REGION Network 2: DESCRIPTION
   // The Energy Efficiency Monitor “EEM” integrated in SICAR is based on the application example in entry ID: 109753230 V1.0 dated 02/2018 of the Siemens Industry Online Support, see: 
   // 
   // https://support.industry.siemens.com/cs/document/109753230/-s7-energy-efficiency-monitor-for-machines?dti=0&lc=en-WW 
   // 
   // **License**  
   // The software package has to be licensed. The necessary license key has to be entered in the data block for energy data “EEmData”, in the array item “licenseKey”. 
   //  
   // {.pageWidth}
   // ![Image](EemEnPiCalc/en/image1.PNG)
   // 
   // The S7 Energy Efficiency-Monitor (or S7 EE-Monitor) allows you to record the energy consumption of your machine in a SIMATIC controller, and to analyze the results on the basis of the energy and media requirements.  
   // https://support.industry.siemens.com/cs/document/109753230/s7-energieeffizienz-monitor-für-maschinen?dti=0&lc=de-WW 
   // 
   // **PLC Data types**  
   //  LSicar_typeEeMenPiCalc 
   //  LSicar_typeEeMenPiEstate 
   //  LSicar_typeEeMenPiLimit 
   //  typeEnMeterOutputData 
   //  typeMeasDataProfileE3 
   //  
   // **WinCC Faceplates**  
   // 
   // ![Image](EemEnPiCalc/en/image3.PNG)
   // 
   // **WinCC Screen**  
   //  
   // ![Image](EemEnPiCalc/en/image4.PNG)
   //  
   // # Devices & networks 
   // 
   // An additional AI Energy Meter has been added and configured in the SICAR project. The user data has been  
   // configured as module version “EE@Industry measured data profile e3”.  
   // 
   // Select the module version according to your requirements. The data assignment in the FC blocks has to be adjusted according to the selected module version. 
   // 
   // ![Image](EemEnPiCalc/en/image5.PNG)
   //  
   //  
   // 
   //  #### PLC Programm blocks 
   // 
   // ##### CallEnSeem  
   // The block is called in OB “CYCLIC_INTERRUPT_100MS_OB” (100ms cycle). The block contains the following instructions which can be found in “Instructions > Optional packages > Energy Suite extensions”.
   // 
   // **EnS_EEm_Calc:**  
   // The instruction calculates operating state-related energy data of machines and plants for uniform efficiency evaluation, in accordance with the VDMA 34179 measuring directive. 
   // 
   // ---
   // Note
   // :     The instruction calculates the energy efficiency value of the respective state for up to 8 operating states, and the global energy efficiency value. 
   // :     The maximum number of configurable measuring points is 10. Refer to the documentation of the entry ID. 
   // 
   // ---
   // 
   // **EnS_EEm_Report:**  
   // The instruction writes the data for the efficiency report to the data log on the SIMATIC memory card, in accordance with the VDMA 34179 measuring directive. The data log is a CSV file. 
   // 
   // ##### CallEnEffMonitor
   // ---
   // Note
   // :     The assignment of the readings as well as the formation of additional signals can be represented only exemplarily here. It has to be adapted to the actual plant conditions! 
   // 
   // ---
   // 
   // * Networks 1 & 2: The readings of the two AI-Energy-Meters are entered in the DB “EeMonitor”, in an array [0..9] in accordance with the measurement data profile “typeMeasDataProfileE3”. 
   // * Network 3: According to the selection of a measuring point on the HMI, data of the respective measuring point is routed to the HMI data area. The selection is done with a Pull-Down menu and a symbolic I/O field. 
   // * Network 4: Several tags in the EnS…data types are not marked as accessible / visible. In order to display these tags on the HMI all the same, they are routed to DB “EeMonitor” in structure “typeEnMeterWorkHmi”. There the tags are marked as accessible / visible.  
   // * Network 5: A collective signal is generated, according to the exemplary calls for OP area 1. This is only an example! The collective signal shows that the plant is producing parts, by a disjunction (OR) of all outputs. If an output is controlled, the plant is moving and producing parts. This collective signal is used later on to generate the energetic states “eState”. A delay of 3 seconds has been configured so that a short break in controlling the outputs will not change the energetic state. *
   // * Network 6: The signals for the energetic states are generated here. 
   // * Network 7: Simulation On/Off: A part counter is simulated here. Note: the simulation can be switched on and off with a button in the screen. 
   // * Network 8: Simulation On/Off. Energy counters for both AI-Energy-Meters are simulated here. Note: the simulation can be switched on and off with a button in the screen. 
   // * Network 9: Call of blocks “EemDemoSimulation” and “EemDemoResetValEMeter”. 
   // * Network 10: Call of block “EemEnPiCalc” and data routing according to the selection of a measuring point on the HMI. 
   // * Network 11: Error evaluation of block “EemEnPiCalc” to generate ProDiag messages. 
   // * Network 12: Error evaluation of block “EnS_EEm_Report” to generate ProDiag messages.  
   // 
   // ##### EemDemoResetValEMeter  
   // 
   // The block resets certain measurement values by controlling the respective outputs in the I/O area of the AI-Energy-Meter. 
   // 
   // ##### EemDemoSimulation  
   // 
   // This block simulates higher or lower energy values, according to the energetic states “eState”. 
   // 
   // ##### EemEnPiCalc
   // This block calculates the ENPI (Energy value Pro Item). It substitutes the script “EEm_EnPI_Efficiency” of the entry ID. 
   // 
   // ---
   // Note
   // :     All block parameters are provided with “pre-defined actual parameters”.
   // 
   // ---
   // 
   // **Operation mode Automatic / Manual**  
   // 
   // The blocks are independent of operation modes. Therefor they are not assigned to any operation mode area. 
   // 
   // **PLC Alarm text list**  
   // 
   // The following PLC alarm text lists have been created: 
   // 
   // * **EEMonitor_Calc_Warn_PD** ProDiag alarm text list for alarms by instruction “EnS_EEm_Calc”.   
   // * **EEMonitor_Report_Warn_PD** ProDiag alarm text list for alarms by instruction “EnS_EEm_Report”.   
   // Both PLC alarm text lists have been entered in the PLC alarm text list “GLOBAL_GENERAL_AlarmTextList”. 
   // 
   // ---
   // Note
   // :     The alarm texts are provided in two languages (German, English). Please consider the multilingual nature of the entries. 
   // 
   // ---
   // 
   // #### PLC Data types 
   // 
   // PLC data types used for PLC program block or HMI faceplate:  
   // ![Image](_Icon/reference.PNG)  See ..\Library Types\LSicar_typeEeMenPiCalc.pdf  
   // 
   // #### WinCC Objects 
   // 
   // **WinCC HMI-tags**  
   // 
   // The HMI tags are stored in the tag table “AI_EnergyMeter_EEM” in the SICAR project.  
   // 
   // **WinCC Text and graphics lists**  
   // 
   // The text list “EE-MONITOR_MEASUREPOINT” contains the texts necessary for the pull-down menu / symbolic I/O field in the screen. Please take into account the multilingual nature of the entries.  
   // 
   // **WinCC Faceplates**  
   // 
   // The faceplates are stored in the project library, in folder “types”. They have been created using several WinCC objects; they are animated depending on the state. 
   // 
   // * EEM_EnPI_EnergyPerItem:	display of ENPI (ENergy Per Item) 
   // * EEM_ViewBar_Diff-AVG-REF:	bar display to compare reference value and average value 
   // * EEM_ViewBar_EState-Total:	bar display of energy status (not used at this time) 
   // * EEM_ViewBarCurve_EState:	Total: bar display and curve display of the energy values  
   // 
   // **WinCC-screen** 
   // 
   // 1. HMI Screens:	EE-MONITOR_ENERGY: display of the energy values 
   // 2. HMI Popup-screens 
   // 	* EEM_LEGEND_Popup: 		Legend 
   // 	* EEM_INFO-MACHINE_Popup: 	Machine information 
   // 	* EEM_STARTMEASURE_Popup: 	Popup to start the normal measurement or the reference measurement  
   // 	* EEM_UIPE_Popup: 		display of voltage, current, power, and energy 
   // 	* MORE_EEM_Popup: 		Popup with additional buttons 
   // 	* MORE_AddOn_Popup: 		supplemented  with button “EE-Monitor” 
   // 
   //  
   // 
   // {.pageWidth}
   // ![Image](EemEnPiCalc/en/image6.PNG)
   //  
   //  
   // 
   // #### Additional information
   // 
   // #### Update info
   // 
   // #### Further documentations
END_REGION

REGION Network 3: select measurement values
   // can be from EnergyMeter driver or directly from any hardware (in this example EnergyMeter module and PAC)
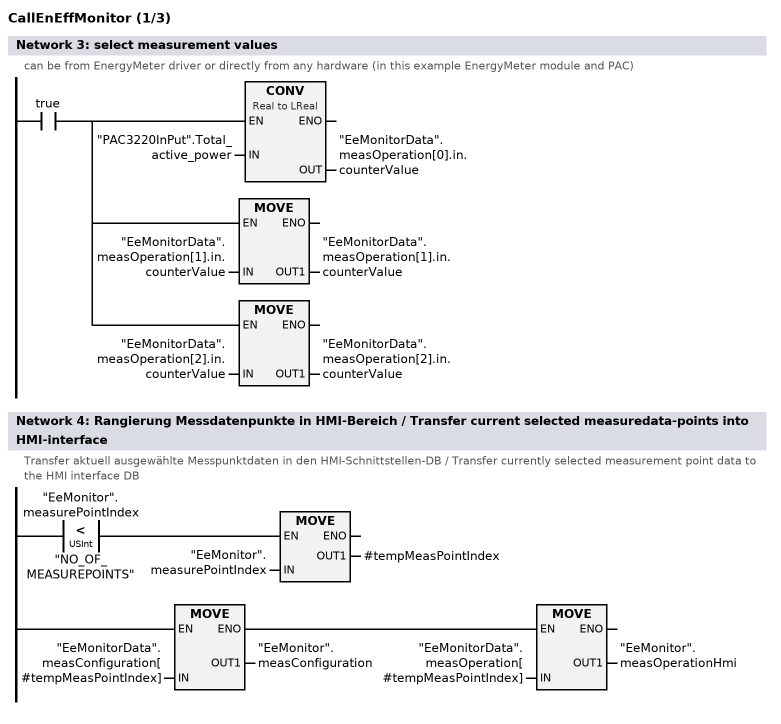
   RUNG wire#powerrail
      Contact( true )
      wire#w1
      { S7_Templates := "[SrcType := Real, DestType := LReal]" } Convert(in := "PAC3220InPut".Total_active_power, out => "EeMonitorData".measOperation[0].in.counterValue)
   END_RUNG
   RUNG wire#w1
      Move(in := "EeMonitorData".measOperation[1].in.counterValue, out1 => "EeMonitorData".measOperation[1].in.counterValue)
   END_RUNG
   RUNG wire#w1
      Move(in := "EeMonitorData".measOperation[2].in.counterValue, out1 => "EeMonitorData".measOperation[2].in.counterValue)
   END_RUNG
   // the same network as SCL:
   IF true THEN
       "EeMonitorData".measOperation[0].in.counterValue := REAL_TO_LREAL("PAC3220InPut".Total_active_power);
       "EeMonitorData".measOperation[1].in.counterValue := "EeMonitorData".measOperation[1].in.counterValue;
       "EeMonitorData".measOperation[2].in.counterValue := "EeMonitorData".measOperation[2].in.counterValue;
   END_IF;
END_REGION

REGION Network 4: Rangierung Messdatenpunkte in HMI-Bereich / Transfer current selected measuredata-points into HMI-interface
   // Transfer aktuell ausgewählte Messpunktdaten in den HMI-Schnittstellen-DB / Transfer currently selected measurement point data to the HMI interface DB
   RUNG wire#powerrail
      { S7_Templates := "SrcType := USInt" } LT_Contact(in1 := "EeMonitor".measurePointIndex, in2 := "NO_OF_MEASUREPOINTS")
      Move(in := "EeMonitor".measurePointIndex, out1 => #tempMeasPointIndex)
   END_RUNG
   RUNG wire#powerrail
      Move(in := "EeMonitorData".measConfiguration[#tempMeasPointIndex], out1 => "EeMonitor".measConfiguration)
      Move(in := "EeMonitorData".measOperation[#tempMeasPointIndex], out1 => "EeMonitor".measOperationHmi)
   END_RUNG
   // the same network as SCL:
   IF "EeMonitor".measurePointIndex < "NO_OF_MEASUREPOINTS" THEN
       #tempMeasPointIndex := "EeMonitor".measurePointIndex;
   END_IF;
   "EeMonitor".measConfiguration := "EeMonitorData".measConfiguration[#tempMeasPointIndex];
   "EeMonitor".measOperationHmi := "EeMonitorData".measOperation[#tempMeasPointIndex];
END_REGION

REGION Network 5: WORKaround: Rangierung / WORKaround: Transfer data from EeMonitroData to EeMonitor.work
   // Konvertierung Zeit in DTL und addieren Zeitzone mit Datum und Uhrzeit aus EnS_EEm_Calc zur Darstellung des tatsächlichen Datums und der tatsächlichen Uhrzeit im aktuellen Land.
   // Convertion of Time to DTL and adding time zone with date and time taken from EnS_EEm_Calc for representing the actual date and time in the current country.
   // Data is copied from EeMonitorData to EeMonitor.work
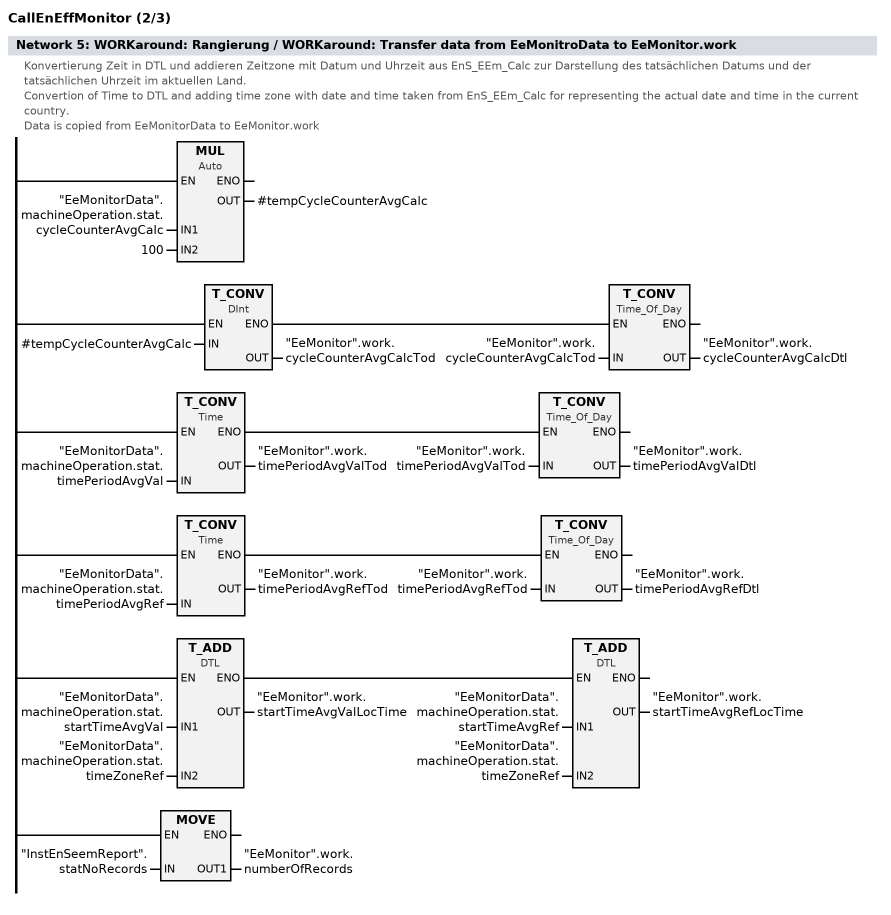
   RUNG wire#powerrail
      Mul(in1 := "EeMonitorData".machineOperation.stat.cycleCounterAvgCalc, in2 := 100, out => #tempCycleCounterAvgCalc)
   END_RUNG
   RUNG wire#powerrail
      { S7_Templates := "[src_type := DInt, dest_type := Time_Of_Day]" } T_CONV(IN := #tempCycleCounterAvgCalc, OUT => "EeMonitor".work.cycleCounterAvgCalcTod)
      { S7_Templates := "[src_type := Time_Of_Day, dest_type := DTL]" } T_CONV(IN := "EeMonitor".work.cycleCounterAvgCalcTod, OUT => "EeMonitor".work.cycleCounterAvgCalcDtl)
   END_RUNG
   RUNG wire#powerrail
      { S7_Templates := "[src_type := Time, dest_type := Time_Of_Day]" } T_CONV(IN := "EeMonitorData".machineOperation.stat.timePeriodAvgVal, OUT => "EeMonitor".work.timePeriodAvgValTod)
      { S7_Templates := "[src_type := Time_Of_Day, dest_type := DTL]" } T_CONV(IN := "EeMonitor".work.timePeriodAvgValTod, OUT => "EeMonitor".work.timePeriodAvgValDtl)
   END_RUNG
   RUNG wire#powerrail
      { S7_Templates := "[src_type := Time, dest_type := Time_Of_Day]" } T_CONV(IN := "EeMonitorData".machineOperation.stat.timePeriodAvgRef, OUT => "EeMonitor".work.timePeriodAvgRefTod)
      { S7_Templates := "[src_type := Time_Of_Day, dest_type := DTL]" } T_CONV(IN := "EeMonitor".work.timePeriodAvgRefTod, OUT => "EeMonitor".work.timePeriodAvgRefDtl)
   END_RUNG
   RUNG wire#powerrail
      { S7_Templates := "[date_type := DTL, time_type := Time]" } T_ADD(IN1 := "EeMonitorData".machineOperation.stat.startTimeAvgVal, IN2 := "EeMonitorData".machineOperation.stat.timeZoneRef, OUT => "EeMonitor".work.startTimeAvgValLocTime)
      { S7_Templates := "[date_type := DTL, time_type := Time]" } T_ADD(IN1 := "EeMonitorData".machineOperation.stat.startTimeAvgRef, IN2 := "EeMonitorData".machineOperation.stat.timeZoneRef, OUT => "EeMonitor".work.startTimeAvgRefLocTime)
   END_RUNG
   RUNG wire#powerrail
      Move(in := "InstEnSeemReport".statNoRecords, out1 => "EeMonitor".work.numberOfRecords)
   END_RUNG
   // the same network as SCL:
   #tempCycleCounterAvgCalc := "EeMonitorData".machineOperation.stat.cycleCounterAvgCalc * 100;
   T_CONV(IN := #tempCycleCounterAvgCalc, OUT => "EeMonitor".work.cycleCounterAvgCalcTod, ENO => #_w1);
   IF #_w1 THEN
       T_CONV(IN := "EeMonitor".work.cycleCounterAvgCalcTod, OUT => "EeMonitor".work.cycleCounterAvgCalcDtl);
   END_IF;
   T_CONV(IN := "EeMonitorData".machineOperation.stat.timePeriodAvgVal,
          OUT => "EeMonitor".work.timePeriodAvgValTod,
          ENO => #_w2);
   IF #_w2 THEN
       T_CONV(IN := "EeMonitor".work.timePeriodAvgValTod, OUT => "EeMonitor".work.timePeriodAvgValDtl);
   END_IF;
   T_CONV(IN := "EeMonitorData".machineOperation.stat.timePeriodAvgRef,
          OUT => "EeMonitor".work.timePeriodAvgRefTod,
          ENO => #_w3);
   IF #_w3 THEN
       T_CONV(IN := "EeMonitor".work.timePeriodAvgRefTod, OUT => "EeMonitor".work.timePeriodAvgRefDtl);
   END_IF;
   T_ADD(IN1 := "EeMonitorData".machineOperation.stat.startTimeAvgVal,
         IN2 := "EeMonitorData".machineOperation.stat.timeZoneRef,
         OUT => "EeMonitor".work.startTimeAvgValLocTime,
         ENO => #_w4);
   IF #_w4 THEN
       T_ADD(IN1 := "EeMonitorData".machineOperation.stat.startTimeAvgRef,
             IN2 := "EeMonitorData".machineOperation.stat.timeZoneRef,
             OUT => "EeMonitor".work.startTimeAvgRefLocTime);
   END_IF;
   "EeMonitor".work.numberOfRecords := "InstEnSeemReport".statNoRecords;
END_REGION

REGION Network 6: Betriebsarten für BA-Bereich1 auf "eState" in "EEm_Data_DB" / Operation modes to "eState"
   // Setzt Estate Nummer abhängig vom ausgewählten OpMode1-Modus / Sets Estate number accoriding to the selected state
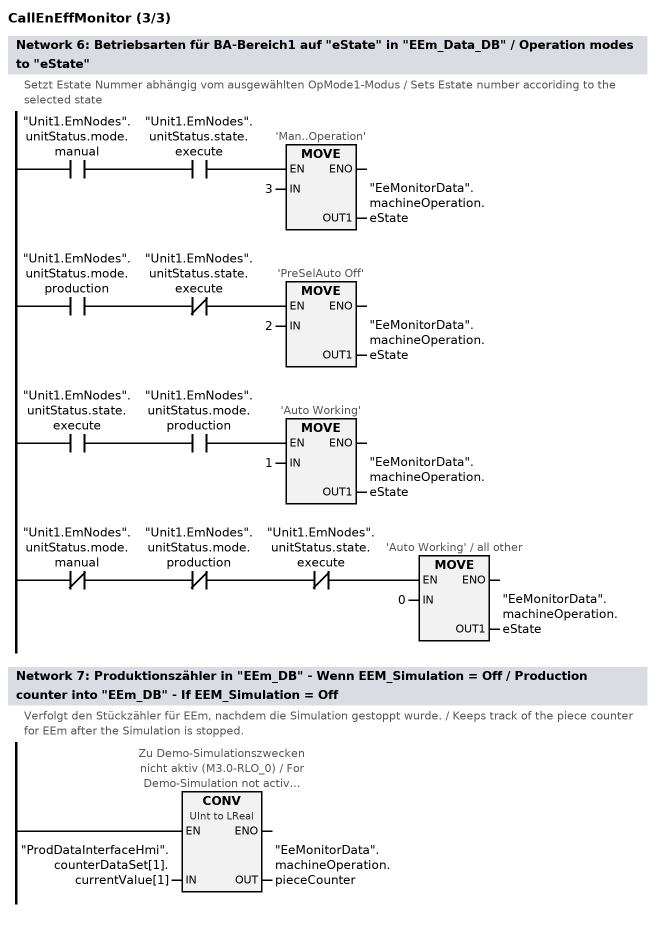
   RUNG wire#powerrail
      Contact( "Unit1.EmNodes".unitStatus.mode.manual )
      Contact( "Unit1.EmNodes".unitStatus.state.execute )
      Move(in := 3, out1 => "EeMonitorData".machineOperation.eState)   // 'Man..Operation'
   END_RUNG
   RUNG wire#powerrail
      Contact( "Unit1.EmNodes".unitStatus.mode.production )
      I_Contact( "Unit1.EmNodes".unitStatus.state.execute )
      Move(in := 2, out1 => "EeMonitorData".machineOperation.eState)   // 'PreSelAuto Off'
   END_RUNG
   RUNG wire#powerrail
      Contact( "Unit1.EmNodes".unitStatus.state.execute )
      Contact( "Unit1.EmNodes".unitStatus.mode.production )
      Move(in := 1, out1 => "EeMonitorData".machineOperation.eState)   // 'Auto Working'
   END_RUNG
   RUNG wire#powerrail
      I_Contact( "Unit1.EmNodes".unitStatus.mode.manual )
      I_Contact( "Unit1.EmNodes".unitStatus.mode.production )
      I_Contact( "Unit1.EmNodes".unitStatus.state.execute )
      Move(in := 0, out1 => "EeMonitorData".machineOperation.eState)   // 'Auto Working' / all other
   END_RUNG
   // the same network as SCL:
   IF "Unit1.EmNodes".unitStatus.mode.manual AND "Unit1.EmNodes".unitStatus.state.execute THEN
       "EeMonitorData".machineOperation.eState := 3;   // 'Man..Operation'
   END_IF;
   IF "Unit1.EmNodes".unitStatus.mode.production AND NOT "Unit1.EmNodes".unitStatus.state.execute THEN
       "EeMonitorData".machineOperation.eState := 2;   // 'PreSelAuto Off'
   END_IF;
   IF "Unit1.EmNodes".unitStatus.state.execute AND "Unit1.EmNodes".unitStatus.mode.production THEN
       "EeMonitorData".machineOperation.eState := 1;   // 'Auto Working'
   END_IF;
   IF NOT "Unit1.EmNodes".unitStatus.mode.manual AND NOT "Unit1.EmNodes".unitStatus.mode.production AND NOT "Unit1.EmNodes".unitStatus.state.execute THEN
       "EeMonitorData".machineOperation.eState := 0;   // 'Auto Working' / all other
   END_IF;
END_REGION

REGION Network 7: Produktionszähler in "EEm_DB" - Wenn EEM_Simulation = Off / Production counter into "EEm_DB" - If EEM_Simulation = Off
   // Verfolgt den Stückzähler für EEm, nachdem die Simulation gestoppt wurde. / Keeps track of the piece counter for EEm after the Simulation is stopped.
   RUNG wire#powerrail
      { S7_Templates := "[SrcType := UInt, DestType := LReal]" } Convert(in := "ProdDataInterfaceHmi".counterDataSet[1].currentValue[1], out => "EeMonitorData".machineOperation.pieceCounter)   // Zu Demo-Simulationszwecken nicht aktiv (M3.0-RLO_0) / For Demo-Simulation not active (M3.0-RLO_0)
   END_RUNG
   // the same network as SCL:
   "EeMonitorData".machineOperation.pieceCounter := UINT_TO_LREAL("ProdDataInterfaceHmi".counterDataSet[1].currentValue[1]);   // Zu Demo-Simulationszwecken nicht aktiv (M3.0-RLO_0) / For Demo-Simulation not active (M3.0-RLO_0)
END_REGION

REGION Network 8 (SCL): Temporary value for storing the EnPi reset time / Reset EnPI values
   // Liest die aktuelle Uhrzeit und speichert sie, um dem Benutzer Informationen über den letzten EnPi-Reset bereitzustellen / Reads the current time and store it to provide the user the information about the last EnPi reset
   // Check for the trigger to reset/recalculate the EnPI values
   IF ("EeMonitorData".internalData.enpiResetTrigger = TRUE) THEN

       // Read the current time and store it to provide the user the information
       // about the last reset
       #tempReturnValue := RD_LOC_T("EeMonitorData".internalData.enpiResetTime);

       // Reset the trigger
       "EeMonitorData".internalData.enpiResetTrigger := FALSE;
   ELSE
       ; // No trigger
   END_IF;
END_REGION
END_FUNCTION

FUNCTION "CallSettings" : Void   // FC8, LAD
// Call of settings blocks
// stored: IsIECCheckEnabled true, SetENOAutomatically false
BEGIN

REGION Network 1: Beschreibung / BLOCK INFO HEADER
   // **Betriebsart Automatik / Hand**  
   // Der Baustein ist keiner Betriebsart / Betriebsartenbereich zugeordnet.  
   // 
   // **Alarme**  
   // Der Baustein generiert keine Alarme.  
   // 
   // #### PLC-Datentypen  
   // Verwendete PLC-Datentypen für den SPS-Programmbaustein und das zugehörige WinCC-Bild.  
   // 
   // {.pageWidth}
   // ![Image](CallInterfaceSignals/de/image1.PNG)
   //  
   //  
   // #### Bausteinaufrufe 
   // Der Baustein “LSicar_InterfaceSignalsBool“ wird in diesem FB als Multi-Instanz aufgerufen, entspr. nebenstehender beispielhafter Darstellung.  
   // 
   // {.pageWidth}
   // ![Image](CallInterfaceSignals/de/image2.PNG)
   //  
   // Um einen neuen FB aufzurufen, ziehen Sie den FB in ein neues Netzwerk, wählen Sie „Multiinstanz“ aus, vergeben Sie einen Namen und parametrieren Sie den FB-Aufruf.  
   // 
   // {.pageWidth}
   // ![Image](CallInterfaceSignals/de/image3.PNG)
   //  
   //  
   // #### Weitere Hinweise 
   // 
   // #### Updateinfo 
   // 
   // #### Weitere Dokumente 
   // 
   // ![Icon](_Icon/reference.PNG)
   // 
   // ..\Library Types\LSicar_InterfaceSignalsBool.pdf
   // SIEMENS AG / (c)Copyright 2023
   // ------------------------------------------------------------------------------
   // Title:            CallSettings
   // Comment/Function: Call of SICAR Settings blocks
   // Library/Family:   -
   // Author:           -
   // Tested with:      ---
   // Engineering:      TIA Portal V19
   // Restrictions:     -
   // Requirements:     ---
   // ------------------------------------------------------------------------------
   // Change log table:
   // Version | Date | Expert in charge | Changes applied
   // -------|---------|-------------|--------------------------------------------
   // 01.00.00 | 01.01.1999 | Person x | First released version
   // 01.00.01 | 02.01.1999 | Person y | Block was Updated
END_REGION

REGION Network 2: Set set PLC date and time
   // Change local date and time of the PLC
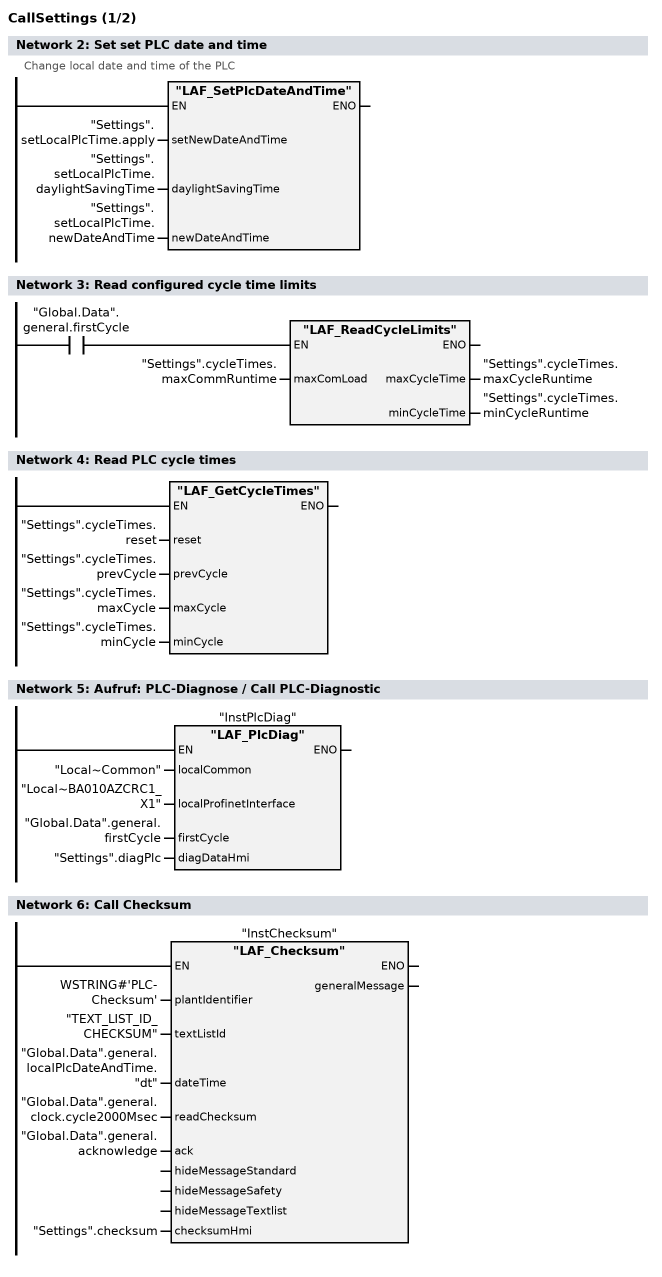
   RUNG wire#powerrail
      "LAF_SetPlcDateAndTime"(setNewDateAndTime := "Settings".setLocalPlcTime.apply, daylightSavingTime := "Settings".setLocalPlcTime.daylightSavingTime, newDateAndTime := "Settings".setLocalPlcTime.newDateAndTime)
   END_RUNG
   // the same network as SCL:
   "LAF_SetPlcDateAndTime"(setNewDateAndTime := "Settings".setLocalPlcTime.apply,
                           daylightSavingTime := "Settings".setLocalPlcTime.daylightSavingTime,
                           newDateAndTime := "Settings".setLocalPlcTime.newDateAndTime);
END_REGION

REGION Network 3: Read configured cycle time limits
   RUNG wire#powerrail
      Contact( "Global.Data".general.firstCycle )
      "LAF_ReadCycleLimits"(maxComLoad := "Settings".cycleTimes.maxCommRuntime, maxCycleTime => "Settings".cycleTimes.maxCycleRuntime, minCycleTime => "Settings".cycleTimes.minCycleRuntime)
   END_RUNG
   // the same network as SCL:
   IF "Global.Data".general.firstCycle THEN
       "LAF_ReadCycleLimits"(maxComLoad := "Settings".cycleTimes.maxCommRuntime,
                             maxCycleTime => "Settings".cycleTimes.maxCycleRuntime,
                             minCycleTime => "Settings".cycleTimes.minCycleRuntime);
   END_IF;
END_REGION

REGION Network 4: Read PLC cycle times
   RUNG wire#powerrail
      "LAF_GetCycleTimes"(reset := "Settings".cycleTimes.reset, prevCycle := "Settings".cycleTimes.prevCycle, maxCycle := "Settings".cycleTimes.maxCycle, minCycle := "Settings".cycleTimes.minCycle)
   END_RUNG
   // the same network as SCL:
   "LAF_GetCycleTimes"(reset := "Settings".cycleTimes.reset,
                       prevCycle := "Settings".cycleTimes.prevCycle,
                       maxCycle := "Settings".cycleTimes.maxCycle,
                       minCycle := "Settings".cycleTimes.minCycle);
END_REGION

REGION Network 5: Aufruf: PLC-Diagnose / Call PLC-Diagnostic
   RUNG wire#powerrail
      "InstPlcDiag"(localCommon := "Local~Common", localProfinetInterface := "Local~BA010AZCRC1_X1", firstCycle := "Global.Data".general.firstCycle, diagDataHmi := "Settings".diagPlc)
   END_RUNG
   // the same network as SCL:
   "InstPlcDiag"(localCommon := "Local~Common",   // "LAF_PlcDiag"
                 localProfinetInterface := "Local~BA010AZCRC1_X1",
                 firstCycle := "Global.Data".general.firstCycle,
                 diagDataHmi := "Settings".diagPlc);
END_REGION

REGION Network 6: Call Checksum
   RUNG wire#powerrail
      "InstChecksum"(plantIdentifier := WSTRING#'PLC-Checksum', textListId := "TEXT_LIST_ID_CHECKSUM", dateTime := "Global.Data".general.localPlcDateAndTime."dt", readChecksum := "Global.Data".general.clock.cycle2000Msec, ack := "Global.Data".general.acknowledge, hideMessageStandard :=, hideMessageSafety :=, hideMessageTextlist :=, checksumHmi := "Settings".checksum, generalMessage =>)
   END_RUNG
   // the same network as SCL:
   "InstChecksum"(plantIdentifier := WSTRING#'PLC-Checksum',   // "LAF_Checksum"
                  textListId := "TEXT_LIST_ID_CHECKSUM",
                  dateTime := "Global.Data".general.localPlcDateAndTime."dt",
                  readChecksum := "Global.Data".general.clock.cycle2000Msec,
                  ack := "Global.Data".general.acknowledge,
                  checksumHmi := "Settings".checksum);
END_REGION

REGION Network 7: Aufruf: SMC-Diagnose (SIMATIC Memory Card - Diagnose) / Call SMC-Diagnostic (SIMATIC Memory Card - Diagnostic)
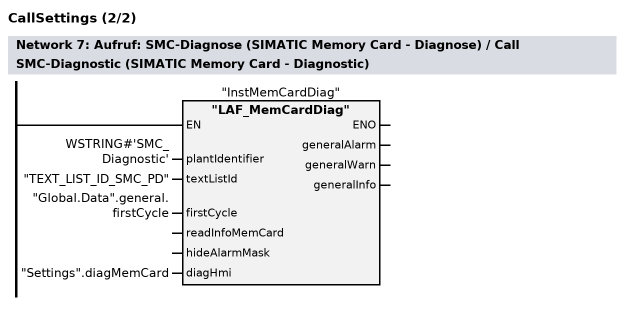
   RUNG wire#powerrail
      "InstMemCardDiag"(plantIdentifier := WSTRING#'SMC_Diagnostic', textListId := "TEXT_LIST_ID_SMC_PD", firstCycle := "Global.Data".general.firstCycle, readInfoMemCard :=, hideAlarmMask :=, diagHmi := "Settings".diagMemCard, generalAlarm =>, generalWarn =>, generalInfo =>)
   END_RUNG
   // the same network as SCL:
   "InstMemCardDiag"(plantIdentifier := WSTRING#'SMC_Diagnostic',   // "LAF_MemCardDiag"
                     textListId := "TEXT_LIST_ID_SMC_PD",
                     firstCycle := "Global.Data".general.firstCycle,
                     diagHmi := "Settings".diagMemCard);
END_REGION
END_FUNCTION

ORGANIZATION_BLOCK "Interrupt1s"   // OB31, LAD, CyclicInterrupt
TITLE = Zyklischer Interrupt 100ms / Cyclic interrupt 100ms
AUTHOR : SICAR
FAMILY : OB
VERSION : 1.0
// organisation block
// stored: IsIECCheckEnabled true, SetENOAutomatically true
   VAR_INPUT
      Initial_Call : Bool;   // Initial call of this OB
      Event_Count : Int;   // Events discarded
   END_VAR
BEGIN

REGION Network 1: Änderungshistorie / ChangeLog
   // Die Änderungshistorie wird nur in englischer Editiersprache geführt.
   // Change log table:
   // Version | Date | Expert in charge | Changes applied
   // -------|---------|-------------|--------------------------------------------
   // 01.00.00 | 01.01.1999 | Person x | First released version
   // 01.00.01 | 02.01.1999 | Person y | Block was Updated
END_REGION

REGION Network 2: EE-MONITOR: Aufruf & Mess-Daten in "EEmData_DB" / Call & measure-data into "EEmData_DB"
   // Aufruf der Energieeffizienz Überwachungs Functionen / Call the energy efficiency monitor functions
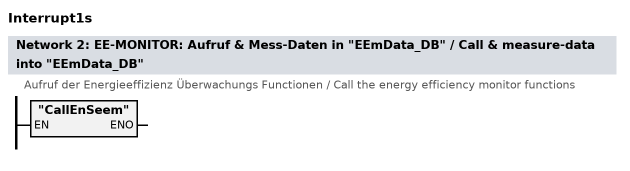
   RUNG wire#powerrail
      "CallEnSeem"()
   END_RUNG
   // the same network as SCL:
   "CallEnSeem"();
END_REGION
END_ORGANIZATION_BLOCK

FUNCTION "CallEnSeem" : Void   // FC34, LAD
TITLE = CallEnSeem
AUTHOR : SICAR
FAMILY : Energy_EEM
VERSION : 1.0
// Der in SICAR eingebaute Energie Effizienz Monitor „EEM“ basiert auf der Beitrags-ID: 109753230, V1.0 von 02/2018 des Siemens Industry Online Support, siehe:  
// https://support.industry.siemens.com/cs/document/109753230/s7-energieeffizienz-monitor-f%C3%BCr-maschinen?dti=0&lc=de-WW  
// 
// **Lizenz**  
// Das Softwarepaket ist Lizenzpflichtig. Die notwendige Lizenz muss im Datenbaustein der Energiedaten „EeMonitorData“ im Datum „licencsKey“ eingetragen werden.  
// 
// 
// Mit dem S7 Energieeffizienz-Monitor können Sie Energieverbräuche Ihrer Maschine in einer SIMATIC Steuerung erfassen und anhand des Energie- und Medienbedarfs statusbezogen anhand der energetischen Zustände analy-sieren. 
//  
//  
// **SPS-Programmbausteine**  
//  
// **PLC-Datentypen**  
//   LSicar_typeEeMenPiCalc  
//   LSicar_typeEeMenPiEstate  
//   LSicar_typeEeMenPiLimit  
//   typeEnMeterOutputData  
//   typeMeasDataProfileE3  
// 
// **WinCC-Bildbaustein**  
//  
// **WinCC-Bild**  
//  
//  
// #### Geräte & Netze
// Im SICAR-Projekt ist ein weiteres AI Energy Meter eingefügt und konfiguriert. Dies ist unter „Nutzdaten“ mit der Modulversion „EE@Industry Messdatenprofil e3“ parametriert.  
// Wählen Sie entsprechend Ihren Anforderungen die Modulversion aus. Je nach gewählter Modulversion, muss die Datenrangierung in den FC-Bausteinen angepasst werden.  
//  
// 
// #### SPS-Programmbausteine
// **CallEnSeem**  
// Der Baustein wird im OB „CYCLIC_INTERRUPT_100MS_OB“ (100ms Takt) aufgerufen. Darin sind nachfolgende Baustein-Anweisungen. Sie sind enthalten unter „Optionspakete > Energy Suite Erweiterungen“.  
// 
// **EnS_EEm_Calc:**  
// Der Baustein berechnet betriebszustandsbezogene Energiedaten von Maschinen und Anlagen zur einheitlichen Effizienzbewertung gemäß Messvorschrift VDMA 34179.  
// 
// NOTE
//  
// :     Der Baustein berechnet für bis zu acht Betriebszustände den Energieeffizienzwert des jeweiligen Zustands sowie den Gesamt-Energieeffizienzwert. 
// :     Die maximale Anzahl der konfigurierbaren Messstellen ist 10. Beachten Sie hierzu die Dokumentation der Beitrags-ID.
// 
// ---
// 
// **EnS_EEm_Report:**  
// Der Baustein erstellt ein Effizienzprotokoll im CSV-Format auf der SIMATIC Memory Card der CPU gemäß Messvorschrift VDMA 34179.  
// 
// **CallEnEffMonitor**  
// 
// NOTE
// :     Die Rangierung der Messdaten, sowie die Bildung von zusätzlichen Signalen kann hier nur beispiel-haft dargestellt werden. Sie muss auf die tatsächlichen Anlagengegebenheiten angepasst werden!
// 
// ---
// 
// * **Netzwerk 1 & 2:** In den beiden Netzwerken werden die Messdaten der beiden AI-Energy-Meter in den DB „EeMonitor“ einge-tragen, in ein Arrayfeld [0..9] gemäß dem Messdatenprofil " typeMeasDataProfileE3".
// * **Netzwerk 3:** Entsprechend des auf dem HMI angewählten Messpunktes (Pull-Down-Menü / Symbolisches E/A-Feld) wer-den hier die Daten des jeweiligen Messpunktes in dem HMI-Datenbereich rangiert.
// * **Netzwerk 4:** Einige Daten in den EnS…-Datentypen (im DB „EeMonitorData“) sind nicht mit Erreichbar/Sichtbar gekenn-zeichnet. Um diese Daten dennoch auf dem HMI darzustellen, werden sie in dem DB „EeMonitor“ rangiert in die Struktur „typeEnMeterWorkHmi“; dort sind die Daten mit Erreichbar/Sichtbar gekennzeichnet. 
// * **Netzwerk 5:** Hier wird ein Summensignal gebildet, entsprechend den Beispiel-Aufrufen für Betriebsartenbereich 1. Es han-delt sich hierbei lediglich um eine Beispiel-Anwendung! Das Summensignal gibt an, das die Anlage Teile pro-duziert. Hierzu werden alle Ausgänge verodert: Werden die Ausgänge angesteuert, so bewegt sich die Anla-ge, die Anlage produziert. Dieses Summensignal wird später benötigt, um damit die energetischen Zustände „eState“ zu bilden. Damit eine kurze Pause bzgl. der Ansteuerung der Ausgänge nicht zu einem Wechsel des energetischen Zustands führt ist hier eine Zeitverzögerung von 3 Sekunden eingebaut.
// * **Netzwerk 6:** In diesem Netzwerk werden die Signale für die energetischen Zustände gebildet.
// * **Netzwerk 7:** Simulation Ein/Aus Betrifft die Simulation von einem Stückzähler. Es wird hier ein simulierter Zähler als Stückzähler verwendet. Hinweis: Die Simulation kann im Bild mittels eines Buttons ein- und ausgeschaltet werden.
// * **Netzwerk 8:** Simulation Ein/Aus Betrifft die Simulation von Energiezähler für beide AI-Energy-Meter. Hinweis: Die Simulation kann im Bild mittels eines Button Ein- und Ausgeschaltet werden.
// * **Netzwerk 9:** Aufruf der Bausteine „EemDemoSimulation“ und „“EemDemoResetValEmeter“.
// * **Netzwerk 10:** Aufruf des Bausteins „EemEnPiCalc“ und Rangierung der daten entspr. dem auf dem HMI ausgewählten Messpunktes.
// * **Netzwerk 11:** Fehlerauswertung des Bausteins “ EemEnPiCalc“ zur Generierung von ProDiag-Meldungen.
// * **Netzwerk 12:** Fehlerauswertung des Bausteins “EnS_EEm_Report“ zur Generierung von ProDiag-Meldungen.
// 
// **EemDemoResetValEmeter** Der Baustein führt ein Reset auf gewisse Messwerte aus, durch Zuweisen der entspr. Ausgänge im E/A-Bereich der AI-Energy-Meter.
// **EemDemoSimulation** Baustein zur Simulation von höheren oder niedrigeren Energiewerten entsprechend der energetischen Zustände „eState“.
// **EemEnPiCalc** Der Baustein berechnet den ENPI (Energiewert Pro Item). Er ersetzt das Skript „EEm_EnPI_Efficiency“ der Bei-trags-ID.
// 
// **Parameter**  
// 
// NOTE
// :     Alle Bausteinparameter sind mit "Vordefinierten Aktualparametern" versehen.
// 
// ---
// 
// **Betriebsart Automatik / Hand** 
// Die Bausteine sind keinem Betriebsartenbereich zugeordnet.  
// 
// **PLC-Meldetextliste**  
// Folgende PLC-Meldetextlisten wurden hierzu angelegt:  
// * EEMonitor_Calc_Warn_PD Beinhaltet die ProDiag-Meldetext für den Bausteinaufruf „EnS_EEm_Calc“.  
// * EEMonitor_Report_Warn_PD Beinhaltet die ProDiag-Meldetexte für den Bausteinaufruf „EnS_EEm_Report“  
// 
// Beide Meldetextlisten sind in der PLC-Meldetextliste „GLOBAL_GENERAL_AlarmTextList“ eingetragen.  
// 
// NOTE
// :    Die Textlisten sind in Deutsch und Englisch ausgeführt. Bitte beachten Sie die Mehrsprachigkeit der PLC-Meldetextlisten.
// 
// ---
// 
// #### PLC-Datentypen
// Verwendete PLC-Datentypen für den SPS-Programmbaustein / WinCC-Bildbaustein:  
// Siehe ..\Library Types\LSicar_typeEeMenPiCalc.pdf  
//  
// #### WinCC-Objekte
// **WinCC HMI-Variablen**  
// Die HMI-Variablen sind im SICAR-Projekt angelegt in der Variablentabelle „AI_EnergyMeter_EEM“  
// 
// **WinCC Text- und Grafiklisten**  
// Die für das im Bild befindliche Pull-Down-Menü / Symbolisches E/A-Feld notwendigen Texte sind in der Text- und Grafikliste „EE-MONITOR_MEASUREPOINT“ hinterlegt. Bitte beachten Sie auch hier die Mehrsprachigkeit.  
// 
// **WinCC-Bildbaustein**  
// Die Bildbausteine befinden sich in der Projekt-Bibliothek unter „Typen“. Sie sind erstellt aus mehreren einzelnen WinCC-Objekten und animiert, je nach Zustand.  
// * EEM_EnPI_EnergyPerItem: Darstellung ENPI (Energy Per Item)
// * EEM_ViewBar_Diff-AVG-REF: Balkendarstellung zum Vergleich zwischen Referenz- / Durchschnittswert
// * EEM_ViewBar_EState-Total: Balkendarstellung Energie Status (z.Zt. nicht verwendet)
// * EEM_ViewBarCurve_EState-Total: Balken- und Kurvendarstellung der Energiewerte
// 
// **WinCC-Bild**  
// * HMI Bilder	
// 	- EE-MONITOR_ENERGY: Darstellung der Energiewerte
// * HMI Popup-Bilder	
// 	- EEM_LEGEND_Popup: Legende
// 	- EEM_INFO-MACHINE_Popup: Maschineninformationen
// 	- EEM_STARTMEASURE_Popup: Popup zum Starten der Normal- oder Referenzmessung
// 	- EEM_UIPE_Popup: Darstellung von Spannung, Strom, Leistung und Energie
// 	- MORE_EEM_Popup: Popup mit zusätzlichen Schaltflächen / Buttons
// 	- MORE_AddOn_Popup: Ergänzt um Button „EE-Monitor“
//  
// #### Weitere Hinweise
// 
// #### Updateinfo
// 
// #### Weitere Dokumente
// The S7 Energy Efficiency-Monitor (or S7 EE-Monitor) allows you to record the energy consumption of your machine in a SIMATIC controller, and to analyze the results on the basis of the energy and media requirements.
// stored: IsIECCheckEnabled true, SetENOAutomatically true
   // Ret_Val : Ret_Val
BEGIN

REGION Network 1: Änderungshistorie / BLOCK INFO HEADER
   // Die Änderungshistorie wird nur in englischer Editiersprache geführt.
   // SIEMENS AG / (c)Copyright 2023
   // ------------------------------------------------------------------------------
   // Title:            CallEnSeem (FC34)
   // Comment/Function: The S7 Energy Efficiency-Monitor (or S7 EE-Monitor) allows you to record the energy consumption of your machine in a SIMATIC controller, and to analyze the results on the basis of the energy and media requirements.
   // Library/Family:   Energy_EEM
   // Author:           SICAR
   // Tested with:      ---
   // Engineering:      TIA Portal V19
   // Restrictions:     -
   // Requirements:     ---
   // ------------------------------------------------------------------------------
   // Change log table:
   // Version | Date | Expert in charge | Changes applied
   // -------|---------|-------------|--------------------------------------------
   // 01.00.00 | 01.01.1999 | Person x | First released version
   // 01.00.01 | 02.01.1999 | Person y | Block was Updated
END_REGION

REGION Network 2: DESCRIPTION
   // The Energy Efficiency Monitor “EEM” integrated in SICAR is based on the application example in entry ID: 109753230 V1.0 dated 02/2018 of the Siemens Industry Online Support, see: 
   // 
   // https://support.industry.siemens.com/cs/document/109753230/-s7-energy-efficiency-monitor-for-machines?dti=0&lc=en-WW 
   // 
   // **License**  
   // The software package has to be licensed. The necessary license key has to be entered in the data block for energy data “EEmData”, in the array item “licenseKey”. 
   //  
   // {.pageWidth}
   // ![Image](EemEnPiCalc/en/image1.PNG)
   // 
   // The S7 Energy Efficiency-Monitor (or S7 EE-Monitor) allows you to record the energy consumption of your machine in a SIMATIC controller, and to analyze the results on the basis of the energy and media requirements.  
   // https://support.industry.siemens.com/cs/document/109753230/s7-energieeffizienz-monitor-für-maschinen?dti=0&lc=de-WW 
   // 
   // **PLC Data types**  
   //  LSicar_typeEeMenPiCalc 
   //  LSicar_typeEeMenPiEstate 
   //  LSicar_typeEeMenPiLimit 
   //  typeEnMeterOutputData 
   //  typeMeasDataProfileE3 
   //  
   // **WinCC Faceplates**  
   // 
   // ![Image](EemEnPiCalc/en/image3.PNG)
   // 
   // **WinCC Screen**  
   //  
   // ![Image](EemEnPiCalc/en/image4.PNG)
   //  
   // # Devices & networks 
   // 
   // An additional AI Energy Meter has been added and configured in the SICAR project. The user data has been  
   // configured as module version “EE@Industry measured data profile e3”.  
   // 
   // Select the module version according to your requirements. The data assignment in the FC blocks has to be adjusted according to the selected module version. 
   // 
   // ![Image](EemEnPiCalc/en/image5.PNG)
   //  
   //  
   // 
   // #### PLC Programm blocks 
   // 
   // ##### CallEnSeem  
   // The block is called in OB “CYCLIC_INTERRUPT_100MS_OB” (100ms cycle). The block contains the following instructions which can be found in “Instructions > Optional packages > Energy Suite extensions”.
   // 
   // **EnS_EEm_Calc:**  
   // The instruction calculates operating state-related energy data of machines and plants for uniform efficiency evaluation, in accordance with the VDMA 34179 measuring directive. 
   // 
   // ---
   // Note
   // :     The instruction calculates the energy efficiency value of the respective state for up to 8 operating states, and the global energy efficiency value. 
   // :     The maximum number of configurable measuring points is 10. Refer to the documentation of the entry ID. 
   // 
   // ---
   // 
   // **EnS_EEm_Report:**  
   // The instruction writes the data for the efficiency report to the data log on the SIMATIC memory card, in accordance with the VDMA 34179 measuring directive. The data log is a CSV file. 
   // 
   // #### CallEnEffMonitor
   // ---
   // Note
   // :     The assignment of the readings as well as the formation of additional signals can be represented only exemplarily here. It has to be adapted to the actual plant conditions! 
   // 
   // ---
   // 
   // * Networks 1 & 2: The readings of the two AI-Energy-Meters are entered in the DB “EeMonitor”, in an array [0..9] in accordance with the measurement data profile “typeMeasDataProfileE3”. 
   // * Network 3: According to the selection of a measuring point on the HMI, data of the respective measuring point is routed to the HMI data area. The selection is done with a Pull-Down menu and a symbolic I/O field. 
   // * Network 4: Several tags in the EnS…data types are not marked as accessible / visible. In order to display these tags on the HMI all the same, they are routed to DB “EeMonitor” in structure “typeEnMeterWorkHmi”. There the tags are marked as accessible / visible.  
   // * Network 5: A collective signal is generated, according to the exemplary calls for OP area 1. This is only an example! The collective signal shows that the plant is producing parts, by a disjunction (OR) of all outputs. If an output is controlled, the plant is moving and producing parts. This collective signal is used later on to generate the energetic states “eState”. A delay of 3 seconds has been configured so that a short break in controlling the outputs will not change the energetic state. *
   // * Network 6: The signals for the energetic states are generated here. 
   // * Network 7: Simulation On/Off: A part counter is simulated here. Note: the simulation can be switched on and off with a button in the screen. 
   // * Network 8: Simulation On/Off. Energy counters for both AI-Energy-Meters are simulated here. Note: the simulation can be switched on and off with a button in the screen. 
   // * Network 9: Call of blocks “EemDemoSimulation” and “EemDemoResetValEMeter”. 
   // * Network 10: Call of block “EemEnPiCalc” and data routing according to the selection of a measuring point on the HMI. 
   // * Network 11: Error evaluation of block “EemEnPiCalc” to generate ProDiag messages. 
   // * Network 12: Error evaluation of block “EnS_EEm_Report” to generate ProDiag messages.  
   // 
   // #### EemDemoResetValEMeter  
   // 
   // The block resets certain measurement values by controlling the respective outputs in the I/O area of the AI-Energy-Meter. 
   // 
   // #### EemDemoSimulation  
   // 
   // This block simulates higher or lower energy values, according to the energetic states “eState”. 
   // 
   // #### EemEnPiCalc
   // This block calculates the ENPI (Energy value Pro Item). It substitutes the script “EEm_EnPI_Efficiency” of the entry ID. 
   // 
   // ---
   // Note
   // :     All block parameters are provided with “pre-defined actual parameters”.
   // 
   // ---
   // 
   // **Operation mode Automatic / Manual**  
   // 
   // The blocks are independent of operation modes. Therefor they are not assigned to any operation mode area. 
   // 
   // **PLC Alarm text list**  
   // 
   // The following PLC alarm text lists have been created: 
   // 
   // * **EEMonitor_Calc_Warn_PD** ProDiag alarm text list for alarms by instruction “EnS_EEm_Calc”.   
   // * **EEMonitor_Report_Warn_PD** ProDiag alarm text list for alarms by instruction “EnS_EEm_Report”.   
   // Both PLC alarm text lists have been entered in the PLC alarm text list “GLOBAL_GENERAL_AlarmTextList”. 
   // 
   // ---
   // Note
   // :     The alarm texts are provided in two languages (German, English). Please consider the multilingual nature of the entries. 
   // 
   // ---
   // 
   // #### PLC Data types 
   // 
   // PLC data types used for PLC program block or HMI faceplate:  
   // ![Image](_Icon/reference.PNG)  See ..\Library Types\LSicar_typeEeMenPiCalc.pdf  
   // 
   // #### WinCC Objects 
   // 
   // **WinCC HMI-tags**  
   // 
   // The HMI tags are stored in the tag table “AI_EnergyMeter_EEM” in the SICAR project.  
   // 
   // **WinCC Text and graphics lists**  
   // 
   // The text list “EE-MONITOR_MEASUREPOINT” contains the texts necessary for the pull-down menu / symbolic I/O field in the screen. Please take into account the multilingual nature of the entries.  
   // 
   // **WinCC Faceplates**  
   // 
   // The faceplates are stored in the project library, in folder “types”. They have been created using several WinCC objects; they are animated depending on the state. 
   // 
   // * EEM_EnPI_EnergyPerItem:	display of ENPI (ENergy Per Item) 
   // * EEM_ViewBar_Diff-AVG-REF:	bar display to compare reference value and average value 
   // * EEM_ViewBar_EState-Total:	bar display of energy status (not used at this time) 
   // * EEM_ViewBarCurve_EState:	Total: bar display and curve display of the energy values  
   // 
   // **WinCC-screen** 
   // 
   // 1. HMI Screens:	EE-MONITOR_ENERGY: display of the energy values 
   // 2. HMI Popup-screens 
   // 	* EEM_LEGEND_Popup: 		Legend 
   // 	* EEM_INFO-MACHINE_Popup: 	Machine information 
   // 	* EEM_STARTMEASURE_Popup: 	Popup to start the normal measurement or the reference measurement  
   // 	* EEM_UIPE_Popup: 		display of voltage, current, power, and energy 
   // 	* MORE_EEM_Popup: 		Popup with additional buttons 
   // 	* MORE_AddOn_Popup: 		supplemented  with button “EE-Monitor” 
   // 
   //  
   // 
   // {.pageWidth}
   // ![Image](EemEnPiCalc/en/image6.PNG)
   //  
   //  
   // 
   // #### Additional information
   // 
   // #### Update info
   // 
   // #### Further documentations
END_REGION

REGION Network 3: EE-Monitor: "Recalc"
   // Toggeln für autom. Aktualisierung der Werte im Bild jeden zweiten Zyklus (alle 200ms) / Toggle for autom. updating the values in the screen every 2nd cycle (every 200ms)
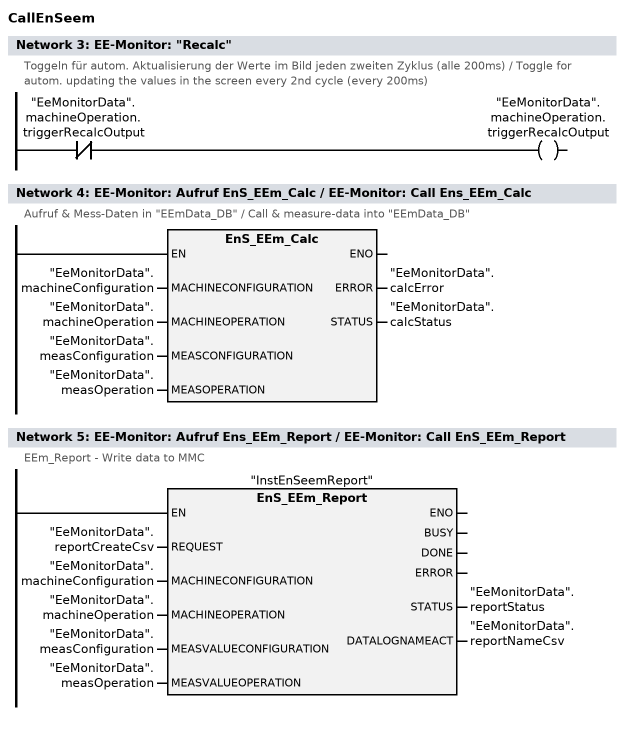
   RUNG wire#powerrail
      I_Contact( "EeMonitorData".machineOperation.triggerRecalcOutput )
      Coil( "EeMonitorData".machineOperation.triggerRecalcOutput )
   END_RUNG
   // the same network as SCL:
   "EeMonitorData".machineOperation.triggerRecalcOutput := NOT "EeMonitorData".machineOperation.triggerRecalcOutput;
END_REGION

REGION Network 4: EE-Monitor: Aufruf EnS_EEm_Calc / EE-Monitor: Call Ens_EEm_Calc
   // Aufruf & Mess-Daten in "EEmData_DB" / Call & measure-data into "EEmData_DB"
   RUNG wire#powerrail
      EnS_EEm_Calc(machineConfiguration := "EeMonitorData".machineConfiguration, machineOperation := "EeMonitorData".machineOperation, measConfiguration := "EeMonitorData".measConfiguration, measOperation := "EeMonitorData".measOperation, error => "EeMonitorData".calcError, status => "EeMonitorData".calcStatus)
   END_RUNG
   // the same network as SCL:
   EnS_EEm_Calc(machineConfiguration := "EeMonitorData".machineConfiguration,
                machineOperation := "EeMonitorData".machineOperation,
                measConfiguration := "EeMonitorData".measConfiguration,
                measOperation := "EeMonitorData".measOperation,
                error => "EeMonitorData".calcError,
                status => "EeMonitorData".calcStatus);
END_REGION

REGION Network 5: EE-Monitor: Aufruf Ens_EEm_Report / EE-Monitor: Call EnS_EEm_Report
   // EEm_Report - Write data to MMC
   RUNG wire#powerrail
      "InstEnSeemReport".EnS_EEm_Report(request := "EeMonitorData".reportCreateCsv, machineConfiguration := "EeMonitorData".machineConfiguration, machineOperation := "EeMonitorData".machineOperation, measValueConfiguration := "EeMonitorData".measConfiguration, measValueOperation := "EeMonitorData".measOperation, busy =>, done =>, error =>, status => "EeMonitorData".reportStatus, dataLogNameAct => "EeMonitorData".reportNameCsv)
   END_RUNG
   // the same network as SCL:
   "InstEnSeemReport"(request := "EeMonitorData".reportCreateCsv,   // EnS_EEm_Report
                      machineConfiguration := "EeMonitorData".machineConfiguration,
                      machineOperation := "EeMonitorData".machineOperation,
                      measValueConfiguration := "EeMonitorData".measConfiguration,
                      measValueOperation := "EeMonitorData".measOperation,
                      status => "EeMonitorData".reportStatus,
                      dataLogNameAct => "EeMonitorData".reportNameCsv);
END_REGION
END_FUNCTION

ORGANIZATION_BLOCK "ProgrammingError"   // OB121, LAD, ProgrammingError
// stored: SetENOAutomatically false
   VAR_INPUT
      BlockNr : UInt;   // Number of causing block
      Reaction : USInt;   // 0:ignore, 1:substitute, 2:skip
      Fault_ID : Byte;   // Fault identifier
      BlockType : USInt;   // 16#01:OB, 16#02:FC, 16#03:FB, 16#04:SFC, 16#05:SFB, 16#06:DB: Type of block causing the error
      Area : USInt;   // Area where the error occured
      DBNr : DB_ANY;   // DB number if Area = DB or DI
      Csg_OBNr : OB_ANY;   // Number of OB causing the error
      Csg_Prio : USInt;   // Priority of OB causing the error
      Width : USInt;   // 0:bit, 1:byte, 2:word, 3:dword, 4:lword
   END_VAR
BEGIN
END_ORGANIZATION_BLOCK

ORGANIZATION_BLOCK "Startup"   // OB100, LAD, Startup
TITLE = "Complete Restart"
// stored: AutoNumber false, IsIECCheckEnabled true, SetENOAutomatically true
   VAR_INPUT
      LostRetentive : Bool;   // True if retentive data are lost
      LostRTC : Bool;   // True if date and time are lost
   END_VAR
   VAR_TEMP
      tempError : Bool;
      tempStatus : Word;
      tempDiagnostics : "LAF_typeDiagnosticsSimple";
   END_VAR
BEGIN

REGION Network 1: Erster Zyklus bit setzen / Set first cycle bit
   // Setze das "erster Zyklus" Signal und die Signale immer EIN sowie immer AUS / Set the first cycle signal
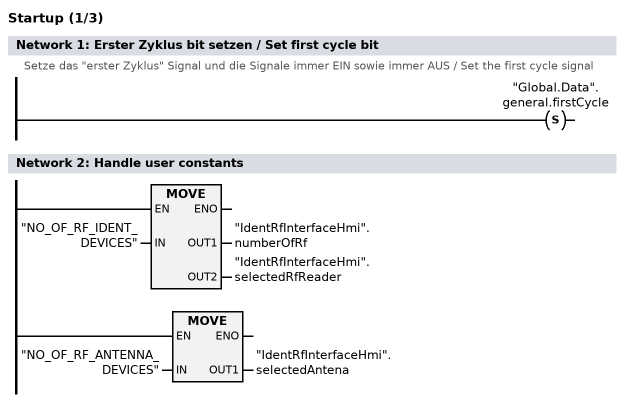
   RUNG wire#powerrail
      S_Coil( "Global.Data".general.firstCycle )
   END_RUNG
   // the same network as SCL:
   "Global.Data".general.firstCycle := TRUE;
END_REGION

REGION Network 2: Handle user constants
   RUNG wire#powerrail
      Move(in := "NO_OF_RF_IDENT_DEVICES", out1 => "IdentRfInterfaceHmi".numberOfRf, out2 => "IdentRfInterfaceHmi".selectedRfReader)
   END_RUNG
   RUNG wire#powerrail
      Move(in := "NO_OF_RF_ANTENNA_DEVICES", out1 => "IdentRfInterfaceHmi".selectedAntena)
   END_RUNG
   // the same network as SCL:
   "IdentRfInterfaceHmi".numberOfRf := "NO_OF_RF_IDENT_DEVICES";
   "IdentRfInterfaceHmi".selectedRfReader := "NO_OF_RF_IDENT_DEVICES";
   "IdentRfInterfaceHmi".selectedAntena := "NO_OF_RF_ANTENNA_DEVICES";
END_REGION

REGION Network 3: Set drive objects for drive diagnostic
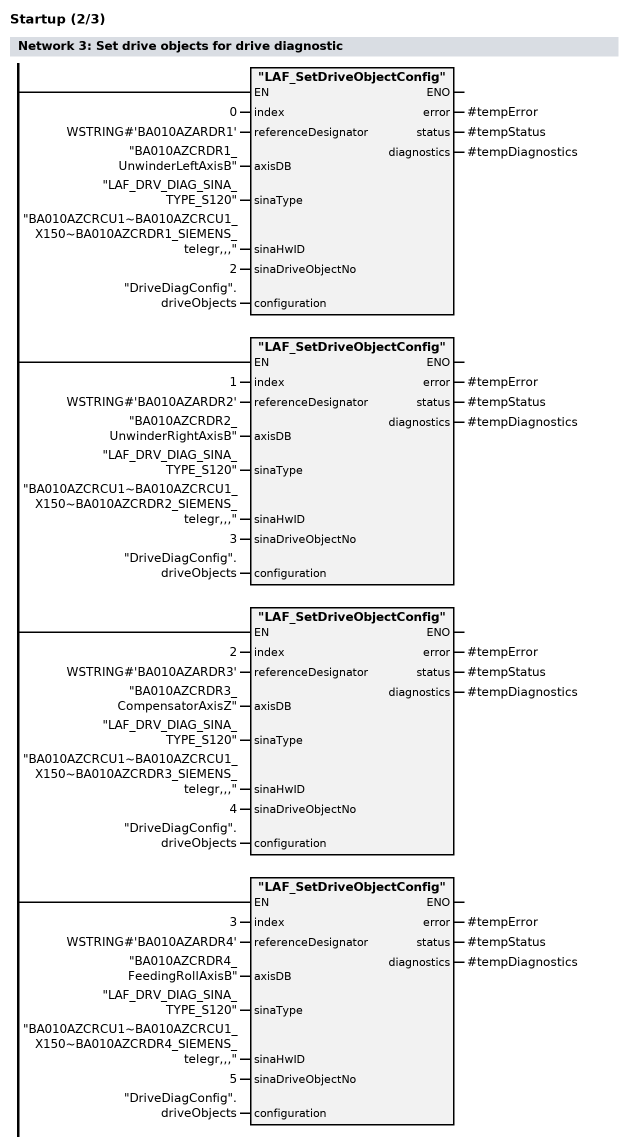
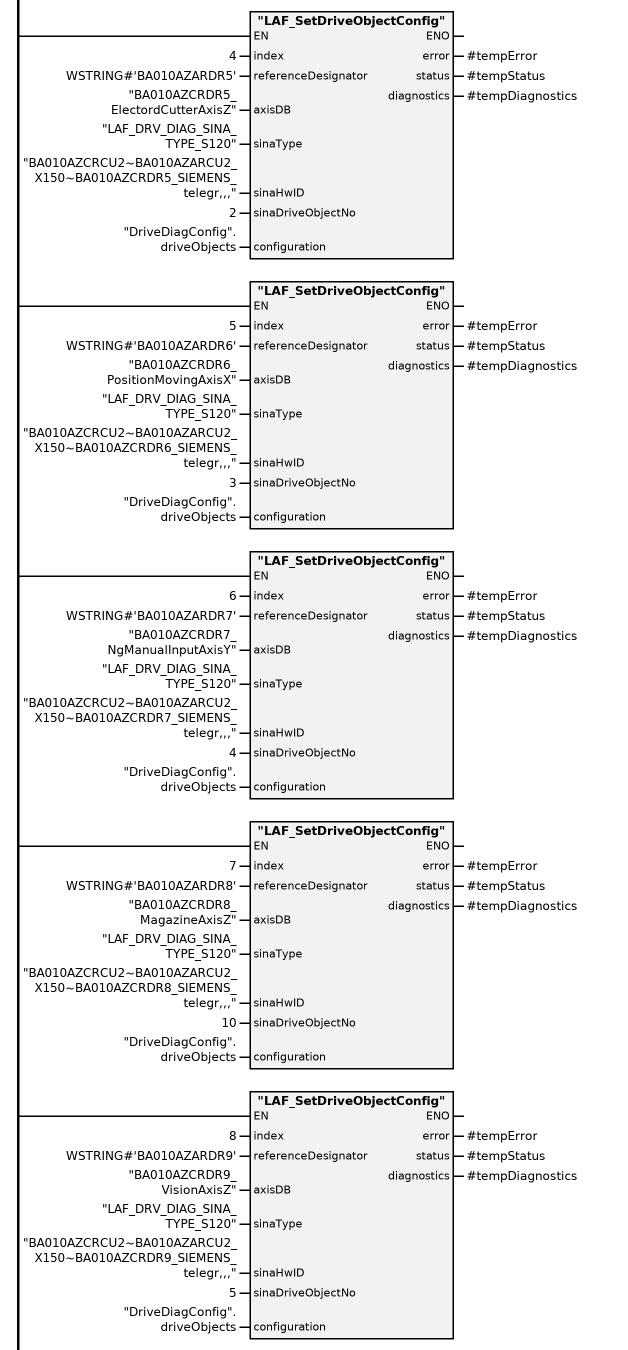
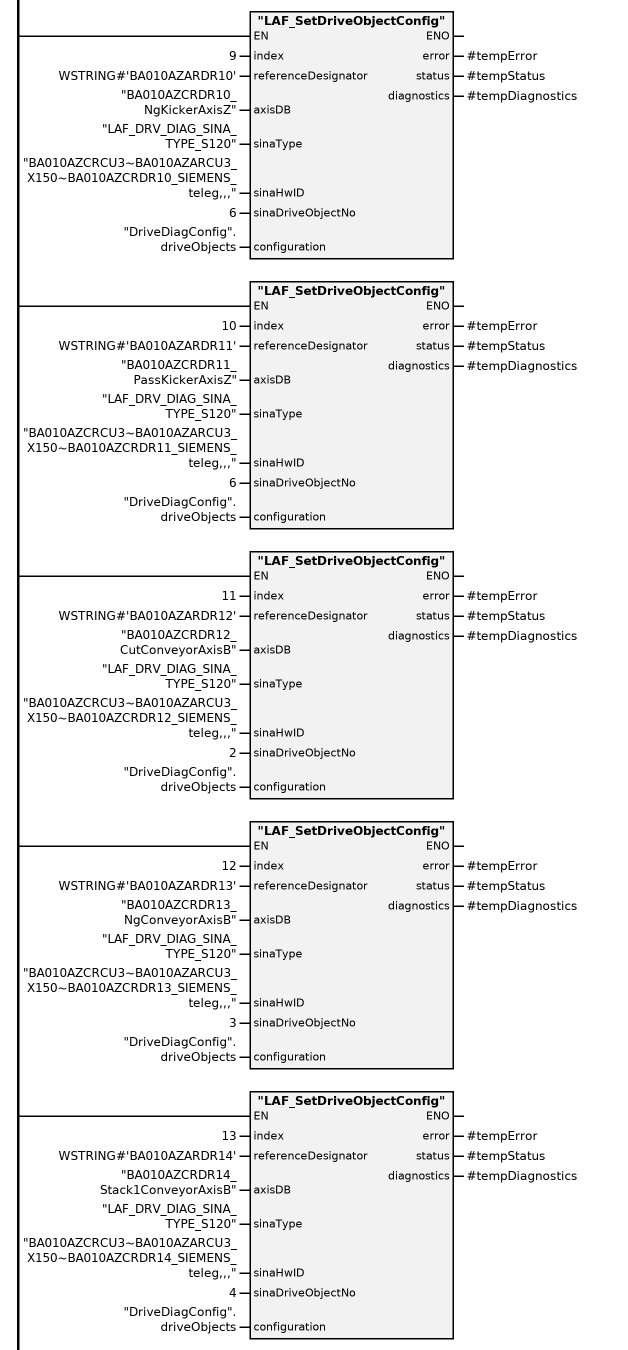
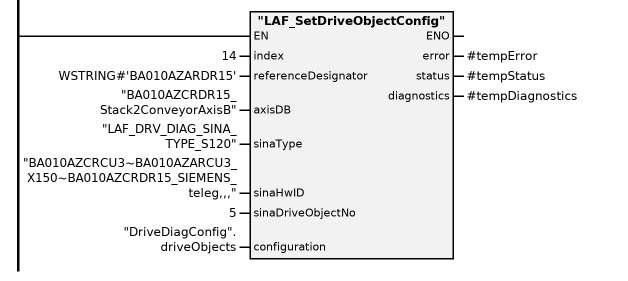
   RUNG wire#powerrail
      "LAF_SetDriveObjectConfig"(index := 0, referenceDesignator := WSTRING#'BA010AZARDR1', axisDB := "BA010AZCRDR1_UnwinderLeftAxisB", sinaType := "LAF_DRV_DIAG_SINA_TYPE_S120", sinaHwID := "BA010AZCRCU1~BA010AZCRCU1_X150~BA010AZCRDR1_SIEMENS_telegr,,,", sinaDriveObjectNo := 2, configuration := "DriveDiagConfig".driveObjects, error => #tempError, status => #tempStatus, diagnostics => #tempDiagnostics)
   END_RUNG
   RUNG wire#powerrail
      "LAF_SetDriveObjectConfig"(index := 1, referenceDesignator := WSTRING#'BA010AZARDR2', axisDB := "BA010AZCRDR2_UnwinderRightAxisB", sinaType := "LAF_DRV_DIAG_SINA_TYPE_S120", sinaHwID := "BA010AZCRCU1~BA010AZCRCU1_X150~BA010AZCRDR2_SIEMENS_telegr,,,", sinaDriveObjectNo := 3, configuration := "DriveDiagConfig".driveObjects, error => #tempError, status => #tempStatus, diagnostics => #tempDiagnostics)
   END_RUNG
   RUNG wire#powerrail
      "LAF_SetDriveObjectConfig"(index := 2, referenceDesignator := WSTRING#'BA010AZARDR3', axisDB := "BA010AZCRDR3_CompensatorAxisZ", sinaType := "LAF_DRV_DIAG_SINA_TYPE_S120", sinaHwID := "BA010AZCRCU1~BA010AZCRCU1_X150~BA010AZCRDR3_SIEMENS_telegr,,,", sinaDriveObjectNo := 4, configuration := "DriveDiagConfig".driveObjects, error => #tempError, status => #tempStatus, diagnostics => #tempDiagnostics)
   END_RUNG
   RUNG wire#powerrail
      "LAF_SetDriveObjectConfig"(index := 3, referenceDesignator := WSTRING#'BA010AZARDR4', axisDB := "BA010AZCRDR4_FeedingRollAxisB", sinaType := "LAF_DRV_DIAG_SINA_TYPE_S120", sinaHwID := "BA010AZCRCU1~BA010AZCRCU1_X150~BA010AZCRDR4_SIEMENS_telegr,,,", sinaDriveObjectNo := 5, configuration := "DriveDiagConfig".driveObjects, error => #tempError, status => #tempStatus, diagnostics => #tempDiagnostics)
   END_RUNG
   RUNG wire#powerrail
      "LAF_SetDriveObjectConfig"(index := 4, referenceDesignator := WSTRING#'BA010AZARDR5', axisDB := "BA010AZCRDR5_ElectordCutterAxisZ", sinaType := "LAF_DRV_DIAG_SINA_TYPE_S120", sinaHwID := "BA010AZCRCU2~BA010AZARCU2_X150~BA010AZCRDR5_SIEMENS_telegr,,,", sinaDriveObjectNo := 2, configuration := "DriveDiagConfig".driveObjects, error => #tempError, status => #tempStatus, diagnostics => #tempDiagnostics)
   END_RUNG
   RUNG wire#powerrail
      "LAF_SetDriveObjectConfig"(index := 5, referenceDesignator := WSTRING#'BA010AZARDR6', axisDB := "BA010AZCRDR6_PositionMovingAxisX", sinaType := "LAF_DRV_DIAG_SINA_TYPE_S120", sinaHwID := "BA010AZCRCU2~BA010AZARCU2_X150~BA010AZCRDR6_SIEMENS_telegr,,,", sinaDriveObjectNo := 3, configuration := "DriveDiagConfig".driveObjects, error => #tempError, status => #tempStatus, diagnostics => #tempDiagnostics)
   END_RUNG
   RUNG wire#powerrail
      "LAF_SetDriveObjectConfig"(index := 6, referenceDesignator := WSTRING#'BA010AZARDR7', axisDB := "BA010AZCRDR7_NgManualInputAxisY", sinaType := "LAF_DRV_DIAG_SINA_TYPE_S120", sinaHwID := "BA010AZCRCU2~BA010AZARCU2_X150~BA010AZCRDR7_SIEMENS_telegr,,,", sinaDriveObjectNo := 4, configuration := "DriveDiagConfig".driveObjects, error => #tempError, status => #tempStatus, diagnostics => #tempDiagnostics)
   END_RUNG
   RUNG wire#powerrail
      "LAF_SetDriveObjectConfig"(index := 7, referenceDesignator := WSTRING#'BA010AZARDR8', axisDB := "BA010AZCRDR8_MagazineAxisZ", sinaType := "LAF_DRV_DIAG_SINA_TYPE_S120", sinaHwID := "BA010AZCRCU2~BA010AZARCU2_X150~BA010AZCRDR8_SIEMENS_telegr,,,", sinaDriveObjectNo := 10, configuration := "DriveDiagConfig".driveObjects, error => #tempError, status => #tempStatus, diagnostics => #tempDiagnostics)
   END_RUNG
   RUNG wire#powerrail
      "LAF_SetDriveObjectConfig"(index := 8, referenceDesignator := WSTRING#'BA010AZARDR9', axisDB := "BA010AZCRDR9_VisionAxisZ", sinaType := "LAF_DRV_DIAG_SINA_TYPE_S120", sinaHwID := "BA010AZCRCU2~BA010AZARCU2_X150~BA010AZCRDR9_SIEMENS_telegr,,,", sinaDriveObjectNo := 5, configuration := "DriveDiagConfig".driveObjects, error => #tempError, status => #tempStatus, diagnostics => #tempDiagnostics)
   END_RUNG
   RUNG wire#powerrail
      "LAF_SetDriveObjectConfig"(index := 9, referenceDesignator := WSTRING#'BA010AZARDR10', axisDB := "BA010AZCRDR10_NgKickerAxisZ", sinaType := "LAF_DRV_DIAG_SINA_TYPE_S120", sinaHwID := "BA010AZCRCU3~BA010AZARCU3_X150~BA010AZCRDR10_SIEMENS_teleg,,,", sinaDriveObjectNo := 6, configuration := "DriveDiagConfig".driveObjects, error => #tempError, status => #tempStatus, diagnostics => #tempDiagnostics)
   END_RUNG
   RUNG wire#powerrail
      "LAF_SetDriveObjectConfig"(index := 10, referenceDesignator := WSTRING#'BA010AZARDR11', axisDB := "BA010AZCRDR11_PassKickerAxisZ", sinaType := "LAF_DRV_DIAG_SINA_TYPE_S120", sinaHwID := "BA010AZCRCU3~BA010AZARCU3_X150~BA010AZCRDR11_SIEMENS_teleg,,,", sinaDriveObjectNo := 6, configuration := "DriveDiagConfig".driveObjects, error => #tempError, status => #tempStatus, diagnostics => #tempDiagnostics)
   END_RUNG
   RUNG wire#powerrail
      "LAF_SetDriveObjectConfig"(index := 11, referenceDesignator := WSTRING#'BA010AZARDR12', axisDB := "BA010AZCRDR12_CutConveyorAxisB", sinaType := "LAF_DRV_DIAG_SINA_TYPE_S120", sinaHwID := "BA010AZCRCU3~BA010AZARCU3_X150~BA010AZCRDR12_SIEMENS_teleg,,,", sinaDriveObjectNo := 2, configuration := "DriveDiagConfig".driveObjects, error => #tempError, status => #tempStatus, diagnostics => #tempDiagnostics)
   END_RUNG
   RUNG wire#powerrail
      "LAF_SetDriveObjectConfig"(index := 12, referenceDesignator := WSTRING#'BA010AZARDR13', axisDB := "BA010AZCRDR13_NgConveyorAxisB", sinaType := "LAF_DRV_DIAG_SINA_TYPE_S120", sinaHwID := "BA010AZCRCU3~BA010AZARCU3_X150~BA010AZCRDR13_SIEMENS_teleg,,,", sinaDriveObjectNo := 3, configuration := "DriveDiagConfig".driveObjects, error => #tempError, status => #tempStatus, diagnostics => #tempDiagnostics)
   END_RUNG
   RUNG wire#powerrail
      "LAF_SetDriveObjectConfig"(index := 13, referenceDesignator := WSTRING#'BA010AZARDR14', axisDB := "BA010AZCRDR14_Stack1ConveyorAxisB", sinaType := "LAF_DRV_DIAG_SINA_TYPE_S120", sinaHwID := "BA010AZCRCU3~BA010AZARCU3_X150~BA010AZCRDR14_SIEMENS_teleg,,,", sinaDriveObjectNo := 4, configuration := "DriveDiagConfig".driveObjects, error => #tempError, status => #tempStatus, diagnostics => #tempDiagnostics)
   END_RUNG
   RUNG wire#powerrail
      "LAF_SetDriveObjectConfig"(index := 14, referenceDesignator := WSTRING#'BA010AZARDR15', axisDB := "BA010AZCRDR15_Stack2ConveyorAxisB", sinaType := "LAF_DRV_DIAG_SINA_TYPE_S120", sinaHwID := "BA010AZCRCU3~BA010AZARCU3_X150~BA010AZCRDR15_SIEMENS_teleg,,,", sinaDriveObjectNo := 5, configuration := "DriveDiagConfig".driveObjects, error => #tempError, status => #tempStatus, diagnostics => #tempDiagnostics)
   END_RUNG
   // the same network as SCL:
   "LAF_SetDriveObjectConfig"(index := 0,
                           referenceDesignator := WSTRING#'BA010AZARDR1',
                           axisDB := "BA010AZCRDR1_UnwinderLeftAxisB",
                           sinaType := "LAF_DRV_DIAG_SINA_TYPE_S120",
                           sinaHwID := "BA010AZCRCU1~BA010AZCRCU1_X150~BA010AZCRDR1_SIEMENS_telegr,,,",
                           sinaDriveObjectNo := 2,
                           configuration := "DriveDiagConfig".driveObjects,
                           error => #tempError,
                           status => #tempStatus,
                           diagnostics => #tempDiagnostics);
   "LAF_SetDriveObjectConfig"(index := 1,
                           referenceDesignator := WSTRING#'BA010AZARDR2',
                           axisDB := "BA010AZCRDR2_UnwinderRightAxisB",
                           sinaType := "LAF_DRV_DIAG_SINA_TYPE_S120",
                           sinaHwID := "BA010AZCRCU1~BA010AZCRCU1_X150~BA010AZCRDR2_SIEMENS_telegr,,,",
                           sinaDriveObjectNo := 3,
                           configuration := "DriveDiagConfig".driveObjects,
                           error => #tempError,
                           status => #tempStatus,
                           diagnostics => #tempDiagnostics);
   "LAF_SetDriveObjectConfig"(index := 2,
                           referenceDesignator := WSTRING#'BA010AZARDR3',
                           axisDB := "BA010AZCRDR3_CompensatorAxisZ",
                           sinaType := "LAF_DRV_DIAG_SINA_TYPE_S120",
                           sinaHwID := "BA010AZCRCU1~BA010AZCRCU1_X150~BA010AZCRDR3_SIEMENS_telegr,,,",
                           sinaDriveObjectNo := 4,
                           configuration := "DriveDiagConfig".driveObjects,
                           error => #tempError,
                           status => #tempStatus,
                           diagnostics => #tempDiagnostics);
   "LAF_SetDriveObjectConfig"(index := 3,
                           referenceDesignator := WSTRING#'BA010AZARDR4',
                           axisDB := "BA010AZCRDR4_FeedingRollAxisB",
                           sinaType := "LAF_DRV_DIAG_SINA_TYPE_S120",
                           sinaHwID := "BA010AZCRCU1~BA010AZCRCU1_X150~BA010AZCRDR4_SIEMENS_telegr,,,",
                           sinaDriveObjectNo := 5,
                           configuration := "DriveDiagConfig".driveObjects,
                           error => #tempError,
                           status => #tempStatus,
                           diagnostics => #tempDiagnostics);
   "LAF_SetDriveObjectConfig"(index := 4,
                           referenceDesignator := WSTRING#'BA010AZARDR5',
                           axisDB := "BA010AZCRDR5_ElectordCutterAxisZ",
                           sinaType := "LAF_DRV_DIAG_SINA_TYPE_S120",
                           sinaHwID := "BA010AZCRCU2~BA010AZARCU2_X150~BA010AZCRDR5_SIEMENS_telegr,,,",
                           sinaDriveObjectNo := 2,
                           configuration := "DriveDiagConfig".driveObjects,
                           error => #tempError,
                           status => #tempStatus,
                           diagnostics => #tempDiagnostics);
   "LAF_SetDriveObjectConfig"(index := 5,
                           referenceDesignator := WSTRING#'BA010AZARDR6',
                           axisDB := "BA010AZCRDR6_PositionMovingAxisX",
                           sinaType := "LAF_DRV_DIAG_SINA_TYPE_S120",
                           sinaHwID := "BA010AZCRCU2~BA010AZARCU2_X150~BA010AZCRDR6_SIEMENS_telegr,,,",
                           sinaDriveObjectNo := 3,
                           configuration := "DriveDiagConfig".driveObjects,
                           error => #tempError,
                           status => #tempStatus,
                           diagnostics => #tempDiagnostics);
   "LAF_SetDriveObjectConfig"(index := 6,
                           referenceDesignator := WSTRING#'BA010AZARDR7',
                           axisDB := "BA010AZCRDR7_NgManualInputAxisY",
                           sinaType := "LAF_DRV_DIAG_SINA_TYPE_S120",
                           sinaHwID := "BA010AZCRCU2~BA010AZARCU2_X150~BA010AZCRDR7_SIEMENS_telegr,,,",
                           sinaDriveObjectNo := 4,
                           configuration := "DriveDiagConfig".driveObjects,
                           error => #tempError,
                           status => #tempStatus,
                           diagnostics => #tempDiagnostics);
   "LAF_SetDriveObjectConfig"(index := 7,
                           referenceDesignator := WSTRING#'BA010AZARDR8',
                           axisDB := "BA010AZCRDR8_MagazineAxisZ",
                           sinaType := "LAF_DRV_DIAG_SINA_TYPE_S120",
                           sinaHwID := "BA010AZCRCU2~BA010AZARCU2_X150~BA010AZCRDR8_SIEMENS_telegr,,,",
                           sinaDriveObjectNo := 10,
                           configuration := "DriveDiagConfig".driveObjects,
                           error => #tempError,
                           status => #tempStatus,
                           diagnostics => #tempDiagnostics);
   "LAF_SetDriveObjectConfig"(index := 8,
                           referenceDesignator := WSTRING#'BA010AZARDR9',
                           axisDB := "BA010AZCRDR9_VisionAxisZ",
                           sinaType := "LAF_DRV_DIAG_SINA_TYPE_S120",
                           sinaHwID := "BA010AZCRCU2~BA010AZARCU2_X150~BA010AZCRDR9_SIEMENS_telegr,,,",
                           sinaDriveObjectNo := 5,
                           configuration := "DriveDiagConfig".driveObjects,
                           error => #tempError,
                           status => #tempStatus,
                           diagnostics => #tempDiagnostics);
   "LAF_SetDriveObjectConfig"(index := 9,
                           referenceDesignator := WSTRING#'BA010AZARDR10',
                           axisDB := "BA010AZCRDR10_NgKickerAxisZ",
                           sinaType := "LAF_DRV_DIAG_SINA_TYPE_S120",
                           sinaHwID := "BA010AZCRCU3~BA010AZARCU3_X150~BA010AZCRDR10_SIEMENS_teleg,,,",
                           sinaDriveObjectNo := 6,
                           configuration := "DriveDiagConfig".driveObjects,
                           error => #tempError,
                           status => #tempStatus,
                           diagnostics => #tempDiagnostics);
   "LAF_SetDriveObjectConfig"(index := 10,
                           referenceDesignator := WSTRING#'BA010AZARDR11',
                           axisDB := "BA010AZCRDR11_PassKickerAxisZ",
                           sinaType := "LAF_DRV_DIAG_SINA_TYPE_S120",
                           sinaHwID := "BA010AZCRCU3~BA010AZARCU3_X150~BA010AZCRDR11_SIEMENS_teleg,,,",
                           sinaDriveObjectNo := 6,
                           configuration := "DriveDiagConfig".driveObjects,
                           error => #tempError,
                           status => #tempStatus,
                           diagnostics => #tempDiagnostics);
   "LAF_SetDriveObjectConfig"(index := 11,
                           referenceDesignator := WSTRING#'BA010AZARDR12',
                           axisDB := "BA010AZCRDR12_CutConveyorAxisB",
                           sinaType := "LAF_DRV_DIAG_SINA_TYPE_S120",
                           sinaHwID := "BA010AZCRCU3~BA010AZARCU3_X150~BA010AZCRDR12_SIEMENS_teleg,,,",
                           sinaDriveObjectNo := 2,
                           configuration := "DriveDiagConfig".driveObjects,
                           error => #tempError,
                           status => #tempStatus,
                           diagnostics => #tempDiagnostics);
   "LAF_SetDriveObjectConfig"(index := 12,
                           referenceDesignator := WSTRING#'BA010AZARDR13',
                           axisDB := "BA010AZCRDR13_NgConveyorAxisB",
                           sinaType := "LAF_DRV_DIAG_SINA_TYPE_S120",
                           sinaHwID := "BA010AZCRCU3~BA010AZARCU3_X150~BA010AZCRDR13_SIEMENS_teleg,,,",
                           sinaDriveObjectNo := 3,
                           configuration := "DriveDiagConfig".driveObjects,
                           error => #tempError,
                           status => #tempStatus,
                           diagnostics => #tempDiagnostics);
   "LAF_SetDriveObjectConfig"(index := 13,
                           referenceDesignator := WSTRING#'BA010AZARDR14',
                           axisDB := "BA010AZCRDR14_Stack1ConveyorAxisB",
                           sinaType := "LAF_DRV_DIAG_SINA_TYPE_S120",
                           sinaHwID := "BA010AZCRCU3~BA010AZARCU3_X150~BA010AZCRDR14_SIEMENS_teleg,,,",
                           sinaDriveObjectNo := 4,
                           configuration := "DriveDiagConfig".driveObjects,
                           error => #tempError,
                           status => #tempStatus,
                           diagnostics => #tempDiagnostics);
   "LAF_SetDriveObjectConfig"(index := 14,
                           referenceDesignator := WSTRING#'BA010AZARDR15',
                           axisDB := "BA010AZCRDR15_Stack2ConveyorAxisB",
                           sinaType := "LAF_DRV_DIAG_SINA_TYPE_S120",
                           sinaHwID := "BA010AZCRCU3~BA010AZARCU3_X150~BA010AZCRDR15_SIEMENS_teleg,,,",
                           sinaDriveObjectNo := 5,
                           configuration := "DriveDiagConfig".driveObjects,
                           error => #tempError,
                           status => #tempStatus,
                           diagnostics => #tempDiagnostics);
END_REGION

REGION Network 4: Manual Operation Line
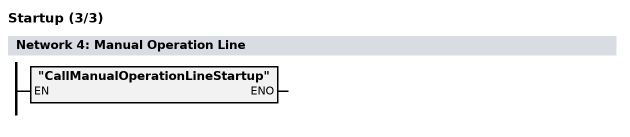
   RUNG wire#powerrail
      "CallManualOperationLineStartup"()
   END_RUNG
   // the same network as SCL:
   "CallManualOperationLineStartup"();
END_REGION
END_ORGANIZATION_BLOCK

FUNCTION "CallManualOperationLineStartup" : Void   // FC99, SCL
// stored: SetENOAutomatically false
BEGIN
   REGION Description
   (*
       Startup call to set the configuration of the Manual Operation Line for the Equipment modules
   *)

   END_REGION

   "LAF_InternalManual".emsWithManualOpConfigured.maxNoOfEms := "NO_OF_EM";

   REGION Unit 1 Equipment Module 0 configuration
       "ManualOperationControl_U1Em0".manualOperationEm.equipmentModuleNum := 1010;
       "ManualOperationControl_U1Em0".manualOperationEmArea[2].displayedLines := '1;';
       "ManualOperationControl_U1Em0".manualOperationEmArea[1].displayedLines := '21-22;';
   END_REGION

   REGION Unit 1 Equipment Module 1 configuration
       "ManualOperationControl_U1Em1".manualOperationEm.equipmentModuleNum := 1020;
       "ManualOperationControl_U1Em1".manualOperationEmArea[2].displayedLines := '1;';
       "ManualOperationControl_U1Em1".manualOperationEmArea[1].displayedLines := '21-22;';
   END_REGION

   REGION Unit 1 Equipment Module 2 configuration
       "ManualOperationControl_U1Em2".manualOperationEm.equipmentModuleNum := 1030;
       "ManualOperationControl_U1Em2".manualOperationEmArea[2].displayedLines := '1';
       "ManualOperationControl_U1Em2".manualOperationEmArea[1].displayedLines := '21-42;';
   END_REGION

   REGION Unit 1 Equipment Module 3 configuration
       "ManualOperationControl_U1Em3".manualOperationEm.equipmentModuleNum := 1040;
       "ManualOperationControl_U1Em3".manualOperationEmArea[2].displayedLines := '1';
       "ManualOperationControl_U1Em3".manualOperationEmArea[1].displayedLines := '21;';
   END_REGION

   REGION Unit 1 Equipment Module 4 configuration
       "ManualOperationControl_U1Em4".manualOperationEm.equipmentModuleNum := 1050;
       "ManualOperationControl_U1Em4".manualOperationEmArea[2].displayedLines := '1-3,11;';
       "ManualOperationControl_U1Em4".manualOperationEmArea[1].displayedLines := '21;';
   END_REGION

   REGION Unit 1 Equipment Module 5 configuration
       "ManualOperationControl_U1Em5".manualOperationEm.equipmentModuleNum := 1060;
       "ManualOperationControl_U1Em5".manualOperationEmArea[2].displayedLines := '11-12;';
       "ManualOperationControl_U1Em5".manualOperationEmArea[1].displayedLines := '21-26;';
   END_REGION

   REGION Unit 1 Equipment Module 6 configuration
       "ManualOperationControl_U1Em6".manualOperationEm.equipmentModuleNum := 1070;
       "ManualOperationControl_U1Em6".manualOperationEmArea[2].displayedLines := '11;';
       "ManualOperationControl_U1Em6".manualOperationEmArea[1].displayedLines := '21;';
   END_REGION

   REGION Unit 1 Equipment Module 7 configuration
       "ManualOperationControl_U1Em7".manualOperationEm.equipmentModuleNum := 1080;
       "ManualOperationControl_U1Em7".manualOperationEmArea[2].displayedLines := '1-6,16-18;';
       "ManualOperationControl_U1Em7".manualOperationEmArea[1].displayedLines := '21;';
   END_REGION

   REGION CITI EM1 configuration
       // Statement section REGION
       "ManualOperationControl_CITIEm1".manualOperationEm.equipmentModuleNum := 5010;
       "ManualOperationControl_CITIEm1".manualOperationEmArea[2].displayedLines := '1-5;';
   END_REGION
END_FUNCTION

FUNCTION "ReadMe01" : Void   // FC7, SCL
// stored: SetENOAutomatically false
BEGIN
   // The folder structure of the software unit CentralFunctions correlates with the main navigation in the HMI.
   // For easier orientation, all folders are listed, but some are empty because there is no PLC logic needed, there is only content on the HMI side.
   // Any PLC logic that should relate to the screens on the HMI for that chapter can be added in this folder.
END_FUNCTION

FUNCTION "ReadMe02" : Void   // FC42, SCL
// stored: SetENOAutomatically false
BEGIN
   // The folder structure of the software unit CentralFunctions correlates with the main navigation in the HMI.
   // For easier orientation, all folders are listed, but some are empty because there is no PLC logic needed, there is only content on the HMI side.
   // Any PLC logic that should relate to the screens on the HMI for that chapter can be added in this folder.
END_FUNCTION

FUNCTION "CallManualOperationLines_ServoCommands" : Void   // FC72, SCL
// stored: SetENOAutomatically false
   VAR_INPUT
      ManualOperationControl : "LBC_typeAxisControlManualCommands";
   END_VAR
   VAR_OUTPUT
      HmiInterface : "LBC_typeAxisControlManualCommands";
   END_VAR
BEGIN
   REGION Commands Mapping
       //#HmiInterface.enableAxis := #ManualOperationControl.enableAxis;
       //#HmiInterface.resetAxis := #ManualOperationControl.resetAxis;

       #HmiInterface.jogForward := #ManualOperationControl.jogForward;
       #HmiInterface.jogBackward := #ManualOperationControl.jogBackward;

       //#HmiInterface.moveVelocity := #ManualOperationControl.moveVelocity;
       //#HmiInterface.stop := #ManualOperationControl.stop;
       //#HmiInterface.posRelative := #ManualOperationControl.posRelative;
       //#HmiInterface.posAbsolute := #ManualOperationControl.posAbsolute;
   END_REGION
END_FUNCTION

FUNCTION "CallManualOperationLines_ServoPos64Commands" : Void   // FC73, SCL
// stored: SetENOAutomatically false
   VAR_INPUT
      ManualOperationControl : "LBC_typeAxis64PosManualCommands";
   END_VAR
   VAR_OUTPUT
      HmiInterface : "LBC_typeAxis64PosManualCommands";
   END_VAR
BEGIN
   REGION Commands Mapping
       //#HmiInterface.enableAxis := #ManualOperationControl.enableAxis;
       //#HmiInterface.resetAxis := #ManualOperationControl.resetAxis;

       #HmiInterface.jogForward := #ManualOperationControl.jogForward;
       #HmiInterface.jogBackward := #ManualOperationControl.jogBackward;

       //#HmiInterface.moveVelocity := #ManualOperationControl.moveVelocity;
       //#HmiInterface.stop := #ManualOperationControl.stop;
       //#HmiInterface.posRelative := #ManualOperationControl.posRelative;
       //#HmiInterface.posAbsolute := #ManualOperationControl.posAbsolute;
   END_REGION
END_FUNCTION

FUNCTION "LAF_ManualOperationLine_Notes" : Void   // FC23, LAD
TITLE = LAF_ManualOperationLine_Notes
// Here are some points that are important for the use and configuration of manual operation lines:
// 
// * For the appearance of each Line, Json files with the configurations need to be added manually to the target machine. Be it in a PC Runtime or Panel. The Path is set in the HMI as the HMI Tag "manualOperationFilePath" in the "03_manualOperation" table. We have set it to "D:\\JsonFiles\\". The files used for this example are saved in the project UserFiles. The Path for the Panel can look like "/home/industrial/JsonFiles".
// 
// * Under "CallManualOperationLines" are the calls for the main configuration of a Equipment module and the control of each line.
//  * Each Equipment module needs to have a defined number. For the numeration we recommend using the second and third digit for the Equipment module number used in the project and the fourth digit with the number of the unit.
// 
// * The texts for the Areas are defined as text lists in the HMI. For the corresponding group, the naming is currently set as "EquipmentAreas_XXXX" with the XXXX as the Equipment Module number. It is set in the "manualOperationEm.equipmentModuleNum".
//  
// * There can be defined 16 color text lists. Each text list defines: "1 - normal, 2 - pressed, 3 - confirmed, 4 - deactivated, 5 - deactivated+pressed".
//  * The color value is in hex with the 2 first values on the left defining the transparency and the rest as normal color values.
//  * The text list name is currently "LAF_manualColorX" with the X as the text list number.
// 
// * If another HMI device is added, please don't forget the Scheduled tasks for updating the lines  
// 
// * The amount of areas is defined by the size of the array in the configuration of areas. The array should start.
// stored: SetENOAutomatically false
BEGIN
END_FUNCTION

FUNCTION "ReadMe04" : Void   // FC11, SCL
// stored: SetENOAutomatically false
BEGIN
   // The folder structure of the software unit CentralFunctions correlates with the main navigation in the HMI.
   // For easier orientation, all folders are listed, but some are empty because there is no PLC logic needed, there is only content on the HMI side.
   // Any PLC logic that should relate to the screens on the HMI for that chapter can be added in this folder.
END_FUNCTION

FUNCTION "ReadMe06" : Void   // FC41, SCL
// stored: SetENOAutomatically false
BEGIN
   // The folder structure of the software unit CentralFunctions correlates with the main navigation in the HMI.
   // For easier orientation, all folders are listed, but some are empty because there is no PLC logic needed, there is only content on the HMI side.
   // Any PLC logic that should relate to the screens on the HMI for that chapter can be added in this folder.
END_FUNCTION

FUNCTION "CallShiftModel" : Void   // FC2, LAD
TITLE = CallShiftModel
// Called LSicar_Shiftmodel
// stored: IsIECCheckEnabled true, SetENOAutomatically true
   VAR_TEMP   // added for the SCL form of the ladder/FBD networks
      _w1 : Bool;
      _w2 : Bool;
      _w3 : Bool;
   END_VAR
BEGIN

REGION Network 1: BLOCK INFO HEADER
   // SIEMENS AG / (c)Copyright 2023
   // ------------------------------------------------------------------------------
   // Title:            CallShiftModel (FC2)
   // Comment/Function: Called LSicar_Shiftmodel 
   // Library/Family:   Automation Framework
   // Author:           Siemens Digital Industry
   // Tested with:      ---
   // Engineering:      TIA Portal V19
   // Restrictions:     -
   // Requirements:     ---
   // ------------------------------------------------------------------------------
   // Change log table:
   // Version  | Date       | Expert in charge       | Changes applied
   // ---------|------------|------------------------|------------------------------
   // 01.00.00 | 11.12.2023 | Siemens Industry Online Support
   //                         First released version
END_REGION

REGION Network 2: Call: shiftmodel
   // FB for handling the shift model and times
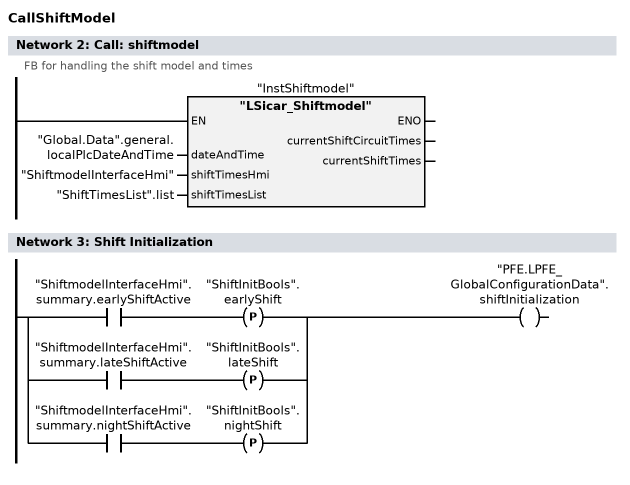
   RUNG wire#powerrail
      "InstShiftmodel"(dateAndTime := "Global.Data".general.localPlcDateAndTime, shiftTimesHmi := "ShiftmodelInterfaceHmi", shiftTimesList := "ShiftTimesList".list, currentShiftCircuitTimes =>, currentShiftTimes =>)
   END_RUNG
   // the same network as SCL:
   "InstShiftmodel"(dateAndTime := "Global.Data".general.localPlcDateAndTime,   // "LSicar_Shiftmodel"
                    shiftTimesHmi := "ShiftmodelInterfaceHmi",
                    shiftTimesList := "ShiftTimesList".list);
END_REGION

REGION Network 3: Shift Initialization
   RUNG wire#powerrail
      Contact( "ShiftmodelInterfaceHmi".summary.earlyShiftActive )
      P_Trig( "ShiftInitBools".earlyShift )
      wire#w1
      Coil( "PFE.LPFE_GlobalConfigurationData".shiftInitialization )
   END_RUNG
   RUNG wire#powerrail
      Contact( "ShiftmodelInterfaceHmi".summary.lateShiftActive )
      P_Trig( "ShiftInitBools".lateShift )
   END_RUNG wire#w1
   RUNG wire#powerrail
      Contact( "ShiftmodelInterfaceHmi".summary.nightShiftActive )
      P_Trig( "ShiftInitBools".nightShift )
   END_RUNG wire#w1
   // the same network as SCL:
   #_w1 := "ShiftmodelInterfaceHmi".summary.earlyShiftActive AND NOT "ShiftInitBools".earlyShift;   // rising edge
   "ShiftInitBools".earlyShift := "ShiftmodelInterfaceHmi".summary.earlyShiftActive;
   #_w2 := "ShiftmodelInterfaceHmi".summary.lateShiftActive AND NOT "ShiftInitBools".lateShift;   // rising edge
   "ShiftInitBools".lateShift := "ShiftmodelInterfaceHmi".summary.lateShiftActive;
   #_w3 := "ShiftmodelInterfaceHmi".summary.nightShiftActive AND NOT "ShiftInitBools".nightShift;   // rising edge
   "ShiftInitBools".nightShift := "ShiftmodelInterfaceHmi".summary.nightShiftActive;
   "PFE.LPFE_GlobalConfigurationData".shiftInitialization := #_w1 OR #_w2 OR #_w3;
END_REGION
END_FUNCTION

FUNCTION "ReadMe10" : Void   // FC44, SCL
// stored: SetENOAutomatically false
BEGIN
   // The folder structure of the software unit CentralFunctions correlates with the main navigation in the HMI.
   // For easier orientation, all folders are listed, but some are empty because there is no PLC logic needed, there is only content on the HMI side.
   // Any PLC logic that should relate to the screens on the HMI for that chapter can be added in this folder.
END_FUNCTION

FUNCTION "ReadMe11" : Void   // FC43, SCL
// stored: SetENOAutomatically false
BEGIN
   // The folder structure of the software unit CentralFunctions correlates with the main navigation in the HMI.
   // For easier orientation, all folders are listed, but some are empty because there is no PLC logic needed, there is only content on the HMI side.
   // Any PLC logic that should relate to the screens on the HMI for that chapter can be added in this folder.
END_FUNCTION

DATA_BLOCK "ShiftmodelInterfaceHmi"   // DB103
TITLE = Schichtzeiten / ShiftmodelTimes
AUTHOR : SICAR
FAMILY : Shiftmodel
VERSION : 1.0
// Global DB fuer Schnittstelle HMI / Global DB for HMI interface
// stored: InstanceOfName LSicar_typeShiftmodelHmi, InstanceOfType UDT
"LSicar_typeShiftmodelHmi"
   // VAR RETAIN
   //    shiftTimesListIndex : DInt;
   //    actualTimesDay : Array[0..7] of "LSicar_typeShiftmodTime1Day";
   //    actualSignalsDay : Array[0..7] of "LSicar_typeShiftmodSign1Day";
   //    summary : "LSicar_typeShiftmodSumHmi";
   //    actualDay : USInt;
   //    shiftTimesListOnOff : Bool := TRUE;   // Schichtzeiten Remote OnOff / Shift times OnOff
   //    setAdjTimes : Bool;
   //    hmiTimesValidFor : Array[0..3] of "LSicar_typeWeekdayBools";
   //    hmiTimes : Array[0..3] of "LSicar_typeShiftmodTime1Shift";   // Schnittstelle Lokale Zeiten (eingeben am HMI) / Interface Local Times (Input on HMI)
   //    productionTimes : "LSicar_typeProdTimesHmi";
   // END_VAR
BEGIN
   hmiTimes[1].endCircuitTime := TOD#05:57:00;
   hmiTimes[2].endCircuitTime := TOD#13:57:00;
   hmiTimes[3].endCircuitTime := TOD#21:57:00;
   hmiTimes[1].start := TOD#06:00:00;
   hmiTimes[2].start := TOD#14:00:00;
   hmiTimes[3].start := TOD#22:00:00;
   hmiTimes[1].break[1].start := TOD#08:00:00;
   hmiTimes[1].break[2].start := TOD#10:00:00;
   hmiTimes[1].break[3].start := TOD#12:00:00;
   hmiTimes[1].break[4].start := TOD#00:00:00;
   hmiTimes[2].break[1].start := TOD#16:00:00;
   hmiTimes[2].break[2].start := TOD#18:00:00;
   hmiTimes[2].break[3].start := TOD#20:00:00;
   hmiTimes[2].break[4].start := TOD#00:00:00;
   hmiTimes[3].break[1].start := TOD#00:00:00;
   hmiTimes[3].break[2].start := TOD#02:00:00;
   hmiTimes[3].break[3].start := TOD#04:00:00;
   hmiTimes[3].break[4].start := TOD#00:00:00;
   hmiTimes[1].break[1].startCircuitTime := TOD#08:02:00;
   hmiTimes[1].break[2].startCircuitTime := TOD#00:00:00;
   hmiTimes[1].break[3].startCircuitTime := TOD#12:02:00;
   hmiTimes[1].break[4].startCircuitTime := TOD#00:00:00;
   hmiTimes[2].break[1].startCircuitTime := TOD#16:02:00;
   hmiTimes[2].break[2].startCircuitTime := TOD#00:00:00;
   hmiTimes[2].break[3].startCircuitTime := TOD#20:02:00;
   hmiTimes[2].break[4].startCircuitTime := TOD#00:00:00;
   hmiTimes[3].break[1].startCircuitTime := TOD#00:02:00;
   hmiTimes[3].break[2].startCircuitTime := TOD#00:00:00;
   hmiTimes[3].break[3].startCircuitTime := TOD#04:02:00;
   hmiTimes[3].break[4].startCircuitTime := TOD#00:00:00;
   hmiTimes[1].break[1].endCircuitTime := TOD#08:13:00;
   hmiTimes[1].break[2].endCircuitTime := TOD#00:00:00;
   hmiTimes[1].break[3].endCircuitTime := TOD#12:13:00;
   hmiTimes[1].break[4].endCircuitTime := TOD#00:00:00;
   hmiTimes[2].break[1].endCircuitTime := TOD#16:13:00;
   hmiTimes[2].break[2].endCircuitTime := TOD#00:00:00;
   hmiTimes[2].break[3].endCircuitTime := TOD#20:13:00;
   hmiTimes[2].break[4].endCircuitTime := TOD#00:00:00;
   hmiTimes[3].break[1].endCircuitTime := TOD#00:13:00;
   hmiTimes[3].break[2].endCircuitTime := TOD#00:00:00;
   hmiTimes[3].break[3].endCircuitTime := TOD#04:13:00;
   hmiTimes[3].break[4].endCircuitTime := TOD#00:00:00;
   hmiTimes[1].break[1].end := TOD#08:15:00;
   hmiTimes[1].break[2].end := TOD#10:10:00;
   hmiTimes[1].break[3].end := TOD#12:15:00;
   hmiTimes[1].break[4].end := TOD#00:00:00;
   hmiTimes[2].break[1].end := TOD#16:15:00;
   hmiTimes[2].break[2].end := TOD#18:10:00;
   hmiTimes[2].break[3].end := TOD#20:15:00;
   hmiTimes[2].break[4].end := TOD#00:00:00;
   hmiTimes[3].break[1].end := TOD#00:15:00;
   hmiTimes[3].break[2].end := TOD#02:10:00;
   hmiTimes[3].break[3].end := TOD#04:15:00;
   hmiTimes[3].break[4].end := TOD#00:00:00;
   hmiTimes[1].end := TOD#13:30:00;
   hmiTimes[2].end := TOD#21:30:00;
   hmiTimes[3].end := TOD#05:30:00;
   hmiTimes[1].startCircuitTime := TOD#13:33:00;
   hmiTimes[2].startCircuitTime := TOD#21:33:00;
   hmiTimes[3].startCircuitTime := TOD#05:33:00;
END_DATA_BLOCK

DATA_BLOCK "InstCallGlobal"   // DB265
// stored: InstanceOfName CallGlobal, InstanceOfType FB
"CallGlobal"
BEGIN
END_DATA_BLOCK

DATA_BLOCK "instTeachingPosMagazineAxisZ"   // DB138
// stored: InstanceOfName LER_TeachingPos_Interface, InstanceOfType FB
"LER_TeachingPos_Interface"
   // VAR_INPUT
   //    enable : Bool;
   //    selectTeachingPos : SInt;
   //    indexTeachingPos : SInt;
   // END_VAR
   // VAR_IN_OUT
   //    configurationSetPositions : Array[0..15] of "LBC_typeAxis64PosSetPosition";
   //    moduleInterface : "LBC_typeAxis64PosInterface";
   //    hmiInterface : Array[0..48] of "LER_TypeTeachingPosInterface";
   // END_VAR
   // VAR
   //    statPulse : Array[0..9] of Bool;
   //    statTonTimer : Array[0..15] of TON_TIME;
   //    statLastTeachingPosIndex : SInt;
   // END_VAR
BEGIN
END_DATA_BLOCK

DATA_BLOCK "instTeachingPosNgAndManualInputAxisY"   // DB129
// stored: InstanceOfName LER_TeachingPos_Interface, InstanceOfType FB
"LER_TeachingPos_Interface"
   // VAR_INPUT
   //    enable : Bool;
   //    selectTeachingPos : SInt;
   //    indexTeachingPos : SInt;
   // END_VAR
   // VAR_IN_OUT
   //    configurationSetPositions : Array[0..15] of "LBC_typeAxis64PosSetPosition";
   //    moduleInterface : "LBC_typeAxis64PosInterface";
   //    hmiInterface : Array[0..48] of "LER_TypeTeachingPosInterface";
   // END_VAR
   // VAR
   //    statPulse : Array[0..9] of Bool;
   //    statTonTimer : Array[0..15] of TON_TIME;
   //    statLastTeachingPosIndex : SInt;
   // END_VAR
BEGIN
END_DATA_BLOCK

DATA_BLOCK "instTeachingPosPositionMovingAxisX"   // DB77
// stored: InstanceOfName LER_TeachingPos_Interface, InstanceOfType FB
"LER_TeachingPos_Interface"
   // VAR_INPUT
   //    enable : Bool;
   //    selectTeachingPos : SInt;
   //    indexTeachingPos : SInt;
   // END_VAR
   // VAR_IN_OUT
   //    configurationSetPositions : Array[0..15] of "LBC_typeAxis64PosSetPosition";
   //    moduleInterface : "LBC_typeAxis64PosInterface";
   //    hmiInterface : Array[0..48] of "LER_TypeTeachingPosInterface";
   // END_VAR
   // VAR
   //    statPulse : Array[0..9] of Bool;
   //    statTonTimer : Array[0..15] of TON_TIME;
   //    statLastTeachingPosIndex : SInt;
   // END_VAR
BEGIN
END_DATA_BLOCK

DATA_BLOCK "instTeachingPosVisionUnitAxisZ"   // DB186
// stored: InstanceOfName LER_TeachingPos_Interface, InstanceOfType FB
"LER_TeachingPos_Interface"
   // VAR_INPUT
   //    enable : Bool;
   //    selectTeachingPos : SInt;
   //    indexTeachingPos : SInt;
   // END_VAR
   // VAR_IN_OUT
   //    configurationSetPositions : Array[0..15] of "LBC_typeAxis64PosSetPosition";
   //    moduleInterface : "LBC_typeAxis64PosInterface";
   //    hmiInterface : Array[0..48] of "LER_TypeTeachingPosInterface";
   // END_VAR
   // VAR
   //    statPulse : Array[0..9] of Bool;
   //    statTonTimer : Array[0..15] of TON_TIME;
   //    statLastTeachingPosIndex : SInt;
   // END_VAR
BEGIN
END_DATA_BLOCK

DATA_BLOCK "instLER_qrHistory_STK1Pos"   // DB306
// stored: InstanceOfName LER_qrHistory, InstanceOfType FB
"LER_qrHistory"
   // VAR_INPUT
   //    trigger : Bool;
   //    commonData : "LER_typeCommonData";
   //    qrData : "LER_typeQrData";
   // END_VAR
   // VAR_IN_OUT
   //    dataHistory : "LER_typeQrHistory";
   // END_VAR
   // VAR
   //    statDeleteData : "LER_typeQrHistory";
   //    statTrigger : Array[0..99] of Bool;
   //    statTonTimer { S7_SetPoint := 'True'} : Array[0..99] of TON_TIME;
   //    statComplete : Array[0..99] of Bool;
   // END_VAR
BEGIN
END_DATA_BLOCK

DATA_BLOCK "instLER_qrHistory_STK2Pos"   // DB307
// stored: InstanceOfName LER_qrHistory, InstanceOfType FB
"LER_qrHistory"
   // VAR_INPUT
   //    trigger : Bool;
   //    commonData : "LER_typeCommonData";
   //    qrData : "LER_typeQrData";
   // END_VAR
   // VAR_IN_OUT
   //    dataHistory : "LER_typeQrHistory";
   // END_VAR
   // VAR
   //    statDeleteData : "LER_typeQrHistory";
   //    statTrigger : Array[0..99] of Bool;
   //    statTonTimer { S7_SetPoint := 'True'} : Array[0..99] of TON_TIME;
   //    statComplete : Array[0..99] of Bool;
   // END_VAR
BEGIN
END_DATA_BLOCK

DATA_BLOCK "instLER_qrHistory_VisionPos"   // DB305
// stored: InstanceOfName LER_qrHistory, InstanceOfType FB
"LER_qrHistory"
   // VAR_INPUT
   //    trigger : Bool;
   //    commonData : "LER_typeCommonData";
   //    qrData : "LER_typeQrData";
   // END_VAR
   // VAR_IN_OUT
   //    dataHistory : "LER_typeQrHistory";
   // END_VAR
   // VAR
   //    statDeleteData : "LER_typeQrHistory";
   //    statTrigger : Array[0..99] of Bool;
   //    statTonTimer { S7_SetPoint := 'True'} : Array[0..99] of TON_TIME;
   //    statComplete : Array[0..99] of Bool;
   // END_VAR
BEGIN
END_DATA_BLOCK

DATA_BLOCK "instLER_visionHistory"   // DB304
// stored: InstanceOfName LER_visionHistory, InstanceOfType FB
"LER_visionHistory"
   // VAR_INPUT
   //    trigger : Bool;
   //    result : "LER_typePartData";
   // END_VAR
   // VAR_IN_OUT
   //    dataHistory : "LER_typeVisionHistory";
   // END_VAR
   // VAR
   //    statDeleteData : "LER_typeVisionHistory";
   //    statTrigger : Array[0..99] of Bool;
   //    statTonTimer { S7_SetPoint := 'True'} : Array[0..99] of TON_TIME;
   //    statComplete : Array[0..99] of Bool;
   // END_VAR
BEGIN
END_DATA_BLOCK

DATA_BLOCK "InstGetAxisStatus"   // DB2
AUTHOR : Siemens Digital Industries
FAMILY : LAF
NAME : LAF_GetAxisStatus
VERSION : 1.1
// stored: InstanceOfName LAF_GetAxisStatus, InstanceOfType FB
"LAF_GetAxisStatus"
   // VAR_INPUT
   //    enable : Bool;
   // END_VAR
   // VAR_OUTPUT
   //    valid { ExternalWritable := 'False'} : Bool;
   //    busy { ExternalWritable := 'False'} : Bool;
   //    error { ExternalWritable := 'False'} : Bool;
   //    status { ExternalWritable := 'False'} : Word;
   //    diagnostics { ExternalWritable := 'False'} : "LAF_typeDiagnostics";
   // END_VAR
   // VAR_IN_OUT
   //    configuration : Array[*] of "LAF_typeDriveDiagConfig";
   //    moduleInterface : "LAF_typeDriveDiagInterfaceHmi";
   // END_VAR
   // VAR
   //    statInternal { ExternalAccessible := 'False'; ExternalVisible := 'False'; ExternalWritable := 'False'} : Struct
   //       enablePrevious : Bool;
   //       valid : Bool;
   //       busy : Bool;
   //       error : Bool;
   //       errorUserCleared : Bool;
   //       errorAutoCleared : Bool;
   //       disablingCompleted : Bool;
   //       diagnostics : "LAF_typeDiagnostics";
   //       emptyDiagnostics : "LAF_typeDiagnostics";
   //    END_STRUCT;
   //    statMainState { ExternalAccessible := 'False'; ExternalVisible := 'False'; ExternalWritable := 'False'} : DInt;
   //    statArrayMin { ExternalAccessible := 'False'; ExternalVisible := 'False'; ExternalWritable := 'False'} : DInt;
   //    statArrayMax { ExternalAccessible := 'False'; ExternalVisible := 'False'; ExternalWritable := 'False'} : DInt;
   // END_VAR
BEGIN
END_DATA_BLOCK

DATA_BLOCK "InstGetSinaAlarms"   // DB74
AUTHOR : Siemens Digital Industries
FAMILY : LAF
NAME : LAF_GetSinaAlarms
VERSION : 1.1
// stored: InstanceOfName LAF_GetSinaAlarms, InstanceOfType FB
"LAF_GetSinaAlarms"
   // VAR_INPUT
   //    enable : Bool;
   // END_VAR
   // VAR_OUTPUT
   //    valid { ExternalWritable := 'False'} : Bool;
   //    busy { ExternalWritable := 'False'} : Bool;
   //    error { ExternalWritable := 'False'} : Bool;
   //    status { ExternalWritable := 'False'} : Word;
   //    diagnostics { ExternalWritable := 'False'} : "LAF_typeDiagnostics";
   //    statusWriteRecord { ExternalWritable := 'False'} : DWord;
   //    statusReadRecord { ExternalWritable := 'False'} : DWord;
   // END_VAR
   // VAR_IN_OUT
   //    configuration : Array[*] of "LAF_typeDriveDiagConfig";
   //    moduleInterface : "LAF_typeDriveDiagInterfaceHmi";
   // END_VAR
   // VAR
   //    statInternal { ExternalAccessible := 'False'; ExternalVisible := 'False'; ExternalWritable := 'False'} : Struct
   //       enablePrevious : Bool;
   //       valid : Bool;
   //       busy : Bool;
   //       error : Bool;
   //       errorUserCleared : Bool;
   //       errorAutoCleared : Bool;
   //       disablingCompleted : Bool;
   //       diagnostics : "LAF_typeDiagnostics";
   //       emptyDiagnostics : "LAF_typeDiagnostics";
   //    END_STRUCT;
   //    statMainState { ExternalAccessible := 'False'; ExternalVisible := 'False'; ExternalWritable := 'False'} : DInt;
   //    statArrayMin { ExternalAccessible := 'False'; ExternalVisible := 'False'; ExternalWritable := 'False'} : DInt;
   //    statArrayMax { ExternalAccessible := 'False'; ExternalVisible := 'False'; ExternalWritable := 'False'} : DInt;
   //    instWriteRecord { ExternalAccessible := 'False'; ExternalVisible := 'False'; ExternalWritable := 'False'} : WRREC;
   //    instReadRecord { ExternalAccessible := 'False'; ExternalVisible := 'False'; ExternalWritable := 'False'} : RDREC;
   //    statWriteReq { ExternalAccessible := 'False'; ExternalVisible := 'False'; ExternalWritable := 'False'} : Struct
   //       header : Struct
   //          reqRef : Byte;
   //          reqID : Byte;
   //          axis : Byte;
   //          noPara : Byte;
   //       END_STRUCT;
   //       data : Array[0..235] of Byte;
   //    END_STRUCT;
   //    statReadReq { ExternalAccessible := 'False'; ExternalVisible := 'False'; ExternalWritable := 'False'} : Struct
   //       header : Struct
   //          reqRef : Byte;
   //          reqID : Byte;
   //          axis : Byte;
   //          noPara : Byte;
   //       END_STRUCT;
   //       data : Array[0..235] of Byte;
   //    END_STRUCT;
   //    instActTimer { ExternalAccessible := 'False'; ExternalVisible := 'False'; ExternalWritable := 'False'} : IEC_TIMER;
   //    instReqTimer { ExternalAccessible := 'False'; ExternalVisible := 'False'; ExternalWritable := 'False'} : IEC_TIMER;
   //    statDataTransRun { ExternalAccessible := 'False'; ExternalVisible := 'False'; ExternalWritable := 'False'} : Bool;
   //    statWriteReqSet { ExternalAccessible := 'False'; ExternalVisible := 'False'; ExternalWritable := 'False'} : Bool;
   //    statActTimerIn { ExternalAccessible := 'False'; ExternalVisible := 'False'; ExternalWritable := 'False'} : Bool;
   //    statPrevTimeValue { ExternalAccessible := 'False'; ExternalVisible := 'False'; ExternalWritable := 'False'} : Time;
   //    statActTimerValueAct { ExternalAccessible := 'False'; ExternalVisible := 'False'; ExternalWritable := 'False'} : Time;
   //    statActTimerValueReq { ExternalAccessible := 'False'; ExternalVisible := 'False'; ExternalWritable := 'False'} : Time;
   //    statPrevDriveIndex { ExternalAccessible := 'False'; ExternalVisible := 'False'; ExternalWritable := 'False'} : DInt;
   // END_VAR
BEGIN
END_DATA_BLOCK

DATA_BLOCK "InstGetSinaEpos"   // DB86
AUTHOR : Siemens Digital Industries
FAMILY : LAF
NAME : LAF_GetSinaEpos
VERSION : 1.1
// stored: InstanceOfName LAF_GetSinaEpos, InstanceOfType FB
"LAF_GetSinaEpos"
   // VAR_INPUT
   //    enable : Bool;
   // END_VAR
   // VAR_OUTPUT
   //    valid { ExternalWritable := 'False'} : Bool;
   //    busy { ExternalWritable := 'False'} : Bool;
   //    error { ExternalWritable := 'False'} : Bool;
   //    status { ExternalWritable := 'False'} : Word;
   //    diagnostics { ExternalWritable := 'False'} : "LAF_typeDiagnostics";
   //    statusWriteRecord { ExternalAccessible := 'False'; ExternalVisible := 'False'; ExternalWritable := 'False'} : DWord;
   //    statusReadRecord { ExternalAccessible := 'False'; ExternalVisible := 'False'; ExternalWritable := 'False'} : DWord;
   // END_VAR
   // VAR_IN_OUT
   //    configuration : Array[*] of "LAF_typeDriveDiagConfig";
   //    moduleInterface : "LAF_typeDriveDiagInterfaceHmi";
   // END_VAR
   // VAR
   //    statInternal { ExternalAccessible := 'False'; ExternalVisible := 'False'; ExternalWritable := 'False'} : Struct
   //       enablePrevious : Bool;
   //       valid : Bool;
   //       busy : Bool;
   //       error : Bool;
   //       errorUserCleared : Bool;
   //       errorAutoCleared : Bool;
   //       disablingCompleted : Bool;
   //       diagnostics : "LAF_typeDiagnostics";
   //       emptyDiagnostics : "LAF_typeDiagnostics";
   //    END_STRUCT;
   //    statMainState { ExternalAccessible := 'False'; ExternalVisible := 'False'; ExternalWritable := 'False'} : DInt;
   //    statArrayMin { ExternalAccessible := 'False'; ExternalVisible := 'False'; ExternalWritable := 'False'} : DInt;
   //    statArrayMax { ExternalAccessible := 'False'; ExternalVisible := 'False'; ExternalWritable := 'False'} : DInt;
   //    instWriteRecord { ExternalAccessible := 'False'; ExternalVisible := 'False'; ExternalWritable := 'False'} : WRREC;
   //    instReadRecord { ExternalAccessible := 'False'; ExternalVisible := 'False'; ExternalWritable := 'False'} : RDREC;
   //    statWriteReq { ExternalAccessible := 'False'; ExternalVisible := 'False'; ExternalWritable := 'False'} : Struct
   //       header : Struct
   //          reqRef : Byte;
   //          reqID : Byte;
   //          axis : Byte;
   //          noPara : Byte;
   //       END_STRUCT;
   //       data : Array[0..235] of Byte;
   //    END_STRUCT;
   //    statReadReq { ExternalAccessible := 'False'; ExternalVisible := 'False'; ExternalWritable := 'False'} : Struct
   //       header : Struct
   //          reqRef : Byte;
   //          reqID : Byte;
   //          axis : Byte;
   //          noPara : Byte;
   //       END_STRUCT;
   //       data : Array[0..235] of Byte;
   //    END_STRUCT;
   //    instActTimer { ExternalAccessible := 'False'; ExternalVisible := 'False'; ExternalWritable := 'False'} : IEC_TIMER;
   //    instReqTimer { ExternalAccessible := 'False'; ExternalVisible := 'False'; ExternalWritable := 'False'} : IEC_TIMER;
   //    statDataTransRun { ExternalAccessible := 'False'; ExternalVisible := 'False'; ExternalWritable := 'False'} : Bool;
   //    statWriteReqSet { ExternalAccessible := 'False'; ExternalVisible := 'False'; ExternalWritable := 'False'} : Bool;
   //    statActTimerIn { ExternalAccessible := 'False'; ExternalVisible := 'False'; ExternalWritable := 'False'} : Bool;
   //    statPrevTimeValue { ExternalAccessible := 'False'; ExternalVisible := 'False'; ExternalWritable := 'False'} : Time;
   //    statActTimerValueAct { ExternalAccessible := 'False'; ExternalVisible := 'False'; ExternalWritable := 'False'} : Time;
   //    statActTimerValueReq { ExternalAccessible := 'False'; ExternalVisible := 'False'; ExternalWritable := 'False'} : Time;
   //    statPrevDriveIndex { ExternalAccessible := 'False'; ExternalVisible := 'False'; ExternalWritable := 'False'} : DInt;
   // END_VAR
BEGIN
END_DATA_BLOCK

